REGION Network 1: Block description — Sections 1 to 2
   // ▄▄▄▄▄▄▄▄▄▄▄▄▄▄▄▄▄▄▄▄▄▄▄▄▄▄▄▄▄▄▄▄▄  ＳＴＡＮＤＡＲＤ  ▄▄ 
   // 
   // 
   // TITLE:    SUBROUTINE — ANALOG OUTPUT SCALE
   // 
   // 
   // ▀▀▀▀▀▀▀▀▀▀▀▀▀▀▀▀▀▀▀▀▀▀▀▀▀▀▀▀▀▀▀▀▀▀▀▀▀▀▀▀▀▀▀▀ 
   // 
   // ┌──────────────────────────────────────────┐
   // │                                          │
   // │          FC18002 — SOFTWARE MODULE DESIGN SPECIFICATION (SMDS)            │
   // │                                          │
   // │      The PDF version of the SMDS for this module is available online here:        │
   // │              https://psop.uk/pal-smds-fc18002-p               │
   // │                                          │
   // │      It is also available as part of the Project User Defined Documentation,      │
   // │      it can be accessed by selecting this module in the Project Tree          │
   // │      (on the left) and pressing SHIFT+F1                        │
   // │                                          │
   // └─────────────────────────────────────── ʷᴵᴰ⁻ᵈᶤᵇ  ┘
   // 
   // FC18001_StdSubScaleAI is a subroutine block that is used to convert a scaled device signal to 
   // an integer signal being passed to an analog output in the form of an output word (QW).
   // 
   // The initial scaled value is a real (floating point) number that matches the calibrated range of 
   // the device in engineering units.
   // 
   // The block monitors the scaled signal to see if the scaled value is out-of-range, the following three 
   // fault signals are generated:
   // 
   // 
   //    •   Over-range (signal is more than a specified percentage above the calibrated 
   //      range of the instrument
   // 
   //    •   Under-range (signal is more than a specified percentage below the calibrated 
   //      range of the instrument
   // 
   //    •   Common out-of-range, either the over-range or under-range fault is active
   // 
   // This is a subroutine block.
   // 
   // 
   // 
   // ▄▄▄▄▄▄▄▄▄▄▄▄▄▄▄▄▄▄▄▄▄▄▄▄▄▄▄▄▄▄▄▄▄▄▄▄▄▄▄▄▄▄▄▄
   // 1.     BLOCK TECHNICAL SUMMARY
   // 
   // 
   //  ――――――――――――――――――――――――――――――――――――――――――
   //  NOMENCLATURE & ADDRESSING
   //  ――――――――――――――――――――――――――――――――――――――――――
   //  BLOCK TITLE         Analog Output Scale
   //  BLOCK FUNCTION GROUP    Subroutine
   //  BLOCK ADDRESS       FC18002
   //  BLOCK SYMBOL        FC18002_StdSubScaleAQ
   //  BLOCK USER ID         StdSubScaleAQ
   // 
   //  ――――――――――――――――――――――――――――――――――――――――――
   //  BLOCK TYPE & USAGE
   //  ――――――――――――――――――――――――――――――――――――――――――
   //  BLOCK TYPE         Function (FC)
   //  BLOCK NUMBER        18002
   //  LANGUAGE           LAD
   //  OPTIMISED ACCESS     Yes
   //  PAL USAGE TYPE       Standard block
   // 
   //  ――――――――――――――――――――――――――――――――――――――――――
   //  METRICS
   //  ――――――――――――――――――――――――――――――――――――――――――
   //  EXECUTION TIME       23.6 μs¹
   //  LOAD MEMORY       30.5 kB
   //  WORK MEMORY           0.5 kB  
   //  ――――――――――――――――――――――――――――――――――――――――――
   //                ¹ Measured on: CPU-1515-2PN (order no. 6ES7512-2AM02-0AB0) 
   //                             https://psop.uk/pal-ds-cpu1515
   // 
   // 
   // 
   // ▂▂▂▂▂▂▂▂▂▂▂▂▂▂▂▂▂▂▂▂▂▂▂▂▂▂▂▂▂▂▂▂▂▂▂▂▂▂▂▂▂▂▂▂
   // Additional document references
   // 
   // 
   // In addition to the documents referenced in OB1 (section DOCUMENT REFERENCES), the 
   // following documents are associated with this module:
   // 
   // 
   //  ――――――――――――――――――――――――――――――――――――――――――
   //  REF.     DOCUMENT NO.       TITLE
   //  ――――――――――――――――――――――――――――――――――――――――――
   //  101  PS2001-5-2312-db00801   DB00802 (analog output raw data) SMDS
   //  102  PS2001-5-2312-db00851   DB00852 (analog output scale data) SMDS
   //  ――――――――――――――――――――――――――――――――――――――――――
   // 
   //                ━━━   ⬙⬙⬙⬙⬙⬙   ━━━
   // 
   // 
   // 
   // ▄▄▄▄▄▄▄▄▄▄▄▄▄▄▄▄▄▄▄▄▄▄▄▄▄▄▄▄▄▄▄▄▄▄▄▄▄▄▄▄▄▄▄▄
   // 1.     FUNCTIONAL DESCRIPTION
   // 
   // 
   // FC18002 is the Analog Output Scale block, it is a subroutine block designed to convert a scaled 
   // signal into a form suitable for an analog output it provides the following broad functions:
   // 
   //    •   Converts a scaled, floating point (real) number that reflects the output range of a 
   //      device, into a raw integer signal for an analog output 
   // 
   //    •   Generate fault signals if the instrument is out of range
   // 
   // 
   // 
   // ▂▂▂▂▂▂▂▂▂▂▂▂▂▂▂▂▂▂▂▂▂▂▂▂▂▂▂▂▂▂▂▂▂▂▂▂▂▂▂▂▂▂▂▂
   // 1.1     Convert a scaled value into an analog output
   // 
   // 
   // The principal function of the block is to convert a scaled, floating point (real) number that reflects 
   // the output range of a device, into a raw integer signal for an analog output (in the form of an 
   // output word, QW).
   // 
   // For example, if a variable speed drive had a scaled operating range of 150 rpm to 1500 rpm and 
   // was driven via a 4-20 mA analog output signal from the PLC, then 4 mA would represent 150 rpm 
   // and 20 mA would represent 1500 rpm.
   // 
   // A typical 4-20 mA analog output signal has a raw value of 0 at 4 mA and 27648 at 20 mA.
   //  
   // The block would generate output values as follows (it would also return every value in between; 
   // five typical values have been shown):
   // 
   // 
   //  ――――――――――――――――――――――――――――――――――――――――――
   //  SCALED OUTPUT SIGNAL   RAW INTEGER VALUE FOR OUTPUT   ACTUAL OUTPUT SIGNAL
   //  ――――――――――――――――――――――――――――――――――――――――――
   //     150.0 rpm                     0              4 MA
   //     487.5 rpm             6,912              8 MA
   //     825.0 rpm           13,824            12 MA
   //      1162.5 rpm           20,736            16 MA
   //      1500.0 rpm           27,648            20 MA
   //  ――――――――――――――――――――――――――――――――――――――――――
   // 
   // 
   // 
   // ▂▂▂▂▂▂▂▂▂▂▂▂▂▂▂▂▂▂▂▂▂▂▂▂▂▂▂▂▂▂▂▂▂▂▂▂▂▂▂▂▂▂▂▂
   // 1.2     Fault signals
   // 
   // 
   // The block is able to generate three fault signals:
   // 
   //    •   Device is over-range
   // 
   //    •   Device is under-range
   // 
   //    •   Device is out-of-range (common signal)
   // 
   // Over-range and under-range faults are generated if the device is reading outside its normal 
   // calibrated range. Over-range if the device is reading higher than its maximum configured value 
   // and under-range if lower than its minimum configured value.
   // 
   // The levels at which the device is considered to be either over-range or under-range (out-of-range), 
   // are set as configurable values passed to the module.
   // 
   // The out-of-range fault signal is a common signal that activates if either the over-range or 
   // under-range signal is 
   // 
   // All three signal activate if there is a configuration error with the data provided to the 
   // module (see § 2.1.2).
   // 
   // 
   // 
   // ▄▄▄▄▄▄▄▄▄▄▄▄▄▄▄▄▄▄▄▄▄▄▄▄▄▄▄▄▄▄▄▄▄▄▄▄▄▄▄▄▄▄▄▄
   // 2.     DETAILED BLOCK DESCRIPTION
   // 
   // 
   // This module, FC18001_StdSubScaleAI is a subroutine block that can be called from other blocks 
   // within the PAL. It is designed to provide a linear conversion of a scaled device output signal in 
   // engineering units (in real format) to an integer value that repre-sents the analog output value 
   // passed to an analog output card (as an integer).
   // 
   // These are the formal module parameters: 
   // 
   // 
   // 
   //  ――――――――――――――――――――――――――――――――――――――――――
   //  PARAM          FUNCTION                      TYPE      IN-OUT 
   //  ――――――――――――――――――――――――――――――――――――――――――
   //  AQ_SCALE_SIGNAL   The scaled value of the device output in       Real      In
   //            engineering units
   // 
   //  AQ_RAW_DATA     Analog output signal configuration data (type,     UT00802    In
   //            range, descriptions card parameters and 
   //            coefficients)
   // 
   //  AQ_SCALE_DATA    Analog output signal scaled value data        UT00852   In
   //            (instrument tag, range, descriptions and 
   //            engineering units)
   // 
   //  AQ_RAW_SIGNAL       The actual analog output             Word     Out
   //            engineering units
   // 
   //  OVER_RANGE       Indicates the scaled signal is above its         Bool      Out
   //            calibrated range by more than the tolerance
   //            value
   // 
   //  UNDER_RANGE     Indicates the scaled signal is below its         Bool      Out
   //            calibrated range by more than the tolerance 
   //            value
   // 
   //  OUT_OF_RANGE      Indicates the scaled signal is outside of its     Bool      Out
   //            calibrated range either over or under range
   //  ――――――――――――――――――――――――――――――――――――――――――
   //  Note:   If a configuration error is present (see § 2.1.2) the three out of range parameters 
   //      will be activated (set true) and the AI_SCALE_SIGNAL signal will be set to zero 
   //      irrespective of the AI_RAW_SIGNAL value.
   // 
   // 
   // The AQ_SCALE_SIGNAL signal is provided directly from the module controlling the device and is 
   // a real number in engineering units (e.g. 1220.4 rpm).
   // 
   // The AQ_RAW_SIGNAL signal is the integer value passed directly to the specific output channel 
   // of the analog output card.
   // 
   // The AQ_RAW_DATA and AQ_SCALE_DATA parameters are UDTs that hold information about the 
   // nature of the AQ_RAW_SIGNAL. In the case of AQ_RAW_DATA it specifies the output type: 
   // voltage, current &c., its range in integer values, various par-ametric information and a textual 
   // description of the signal. In the case of AQ_SCALE_DATA it specifies the scaled range of the 
   // signal, its engineering units, out-of-range values, a textual description of the device and the 
   // device tag itself.
   // 
   // 
   //  ――――――――――――――――――――――――――――――――――――――――――
   //  PARAM         ASSOCIATED UDT            ASSOCIATED DATA BLOCK
   //  ――――――――――――――――――――――――――――――――――――――――――
   //  AQ_RAW_DATA    UT00802_St_ConstAqRawData     DB00802_St_ConstAqRawData
   //  AQ_SCALE_DATA   UT00852_St_ConstAqScaleData      DB00852_St_ConstAqScaleData
   //  ――――――――――――――――――――――――――――――――――――――――――
   // 
   // Section 2.1.1 contains a full description of the AQ_RAW_DATA and AQ_SCALE_DATA parameters.
   // 
   // AQ_SCALE_SIGNAL is the true scaled value of the signal being passed to the analog output 
   // (AQ_RAW_SIGNAL) in engineering units.
   // 
   // OVER_RANGE and UNDER_RANGE indicate if the scaled signal is outside its permitted range. 
   // The limits at which under-range and over-range faults activate are provided as part of the 
   // information supplied via the AQ_SCALE_DATA parameter.
   // 
   // OVER_RANGE indicates the output is higher than the permitted tolerance and UNDER_RANGE 
   // indicates the output is lower than the permitted tolerance.
   // 
   // OUT_OF_RANGE is simply a common signal indicating the either OVER_RANGE or UNDER_RANGE 
   // is active.
   // 
   // This arrangement conforms with the PAL philosophy where IO card connections, safety signals 
   // and interlocks have unique formal parameters; all remaining signals are passed as variables 
   // within UDTs, see the Software Design Specification [Ref 008].
   // 
   // 
   // 
   // ▂▂▂▂▂▂▂▂▂▂▂▂▂▂▂▂▂▂▂▂▂▂▂▂▂▂▂▂▂▂▂▂▂▂▂▂▂▂▂▂▂▂▂▂
   // 2.1     Converting the scaled device signal to an analog output value
   // 
   // 
   // The AQ_RAW_SIGNAL is the raw device signal passed to the analog output card; this has specific 
   // ranges depending on the type of IO card and the type of signal in use. 
   //  
   // The following table shows example ranges for the AI_RAW_SIGNAL signal:
   // 
   //  ―――――――――――――――――――――――――――――――――――――――――― 
   //             LOWER LIMIT    EQUIVALENT UPPER LIMIT   EQUIVALENT
   //  SIGNAL TYPE      (RAW_MIN)         TO    (RAW_MAX)       TO      
   //  ―――――――――――――――――――――――――――――――――――――――――― 
   //  -10 V to 10 V         -27648     -10 V        27648      +10 V      
   //  0 V to 10 V          0       +10 V     27648      +10 V      
   //  1 V to 5 V          0      +1 V        27648     +5 V      
   //  -20 mA to 20 mA       -27648     -20 mA    27648      +20 mA      
   //  0 mA to 20 mA         0        0 mA    27648      +20 mA      
   //  4 mA to 20 mA (2/4w)      0        4 mA    27648      +20 mA      
   //  ――――――――――――――――――――――――――――――――――――――――――
   //  Example ranges for an analog output signal
   // 
   // 
   // The RAW_MIN and the RAW_MAX values in the above tables are the numerical values for the 
   // analog output range; the appropriate values are supplied as the RAW_MIN and RAW_MAX 
   // variables provided in the UDT of parameter AQ_RAW_DATA. (see § 2.1.1 for a full description).
   // 	
   // 
   // The corresponding values for the originating scaled device signal are similarly provided by the 
   // SCALE_MIN and SCALE_MAX values provided in the UDT of parameter AQ_SCALE_DATA 
   // (see § 2.1.1 for a full description).
   // 
   // Thus, if a variable speed drive had a scaled operating range of 150 rpm to 1500 rpm that was 
   // passed from the PLC as a 4 20 mA signal, 
   // 
   // 
   //  ――――――――――――――――――――――――――――――――――――――――――
   //  SIGNAL NAME            FUNCTION                   VALUE
   //  ――――――――――――――――――――――――――――――――――――――――――
   //  AQ_RAW_DATA.RAW_MIN     RANGE — Minimum value of the raw analog      0
   //                       signal (at the card)
   //  AQ_RAW_DATA.RAW_MAX    RANGE — Maximum value of the raw analog        27648
   //                       signal (at the card)
   //  AQ_SCALE_DATA.SCALE_MIN   RANGE — Minimum value of the scaled analog       150 rpm
   //                       signal [engineering units]
   //  AQ_SCALE_DATA.SCALE_MAX  RANGE — Maximum value of the scaled analog      1500 rpm
   //                       signal [engineering units]
   //  ――――――――――――――――――――――――――――――――――――――――――
   // 
   // The scaled value from the originating device is passed to the module as a real number in the 
   // parameter: AQ_SCALE_SIGNAL
   // 
   // The analog output signal (AQ_RAW_SIGNAL) is calculated as follows:
   // 
   // 
   // ┌────────────────────────────────────────────┐
   // │                                 (AQ_SCALE_SIGNAL ─ SCALE_MIN) ╳ (RAW_MAX ─ RAW_MIN)         │
   // │AQ_RAW_SIGNAL =  ――――――――――――――――――――――――――――  ┼ RAW_MIN      │
   // │                                    (SCALE_MAX ─ SCALE_MIN)                  │
   // └──────────────────────────────────────  (2.1)  ───┘
   // 
   // In the above calculation, RAW_MIN and RAW_MAX are preceded by AQ_RAW_DATA. and SCALE_MIN and 
   // SCALE_MAX are preceded by AQ_SCALE_DATA.
   // 
   // The three signals: AQ_SCALE_SIGNAL, SCALE_MIN and SCALE_MAX are all floating-point numbers 
   // (real data type), the signals AQ_RAW_SIGNAL, RAW_MIN and RAW_MAX are all integers (int data type).
   // 
   // Note:    It is assumed that the instrument has a linear response.
   // 
   // 
   //           AQ_ SCALE_VALUE
   //             ↑                    ⋰
   //            SCALE_MAX__│______________________________________⋰
   //             │                  ╱|
   //             │                 ╱ |     
   //             │                ╱  |
   //             │               ╱   |
   //             │              ╱    |
   //             │             ╱     |
   //             │            ╱      |
   //     AQ_SCALE_SIGNAL │- - - - - - - - - - - - - - - - - - - - -> ╱       |
   //             │          ╱╎          |
   //             │         ╱ ╎       |
   //             │        ╱  ╎       |
   //             │       ╱   ╎       |   
   //             │      ╱    ╎       |
   //             │     ╱     ╎       |
   //             │    ╱         ╎          |
   //             SCALE_MIN__│______╱          ╎          |
   //             │  ⋰|           ╎          |
   //             │ ⋰ |           ↓          |
   //             ┼─────────────────────────→ AQ_RAW_SIGNAL
   //                   |           ╎           |
   //                RAW_MIN        ╎        RAW_MAX
   //                       AQ_RAW_SIGNAL
   // 
   //    Figure 2.1    Linear relationship between AQ_SCALE_SIGNAL and AQ_RAW_SIGNAL
   // 
   // 
   // 
   // ▁▁▁▁▁▁▁▁▁▁▁▁▁▁▁▁▁▁▁▁▁▁▁▁▁▁▁▁▁▁▁▁▁▁▁▁▁▁▁▁▁▁▁▁
   // 2.1.1     Using AQ_RAW_DATA and AQ_SCALE_DATA
   // 
   // 
   // 
   // ▁▁▁▁▁▁▁▁▁▁▁▁▁▁▁▁▁▁▁▁▁▁▁▁▁▁▁▁▁▁▁▁▁▁▁▁▁▁▁▁▁▁▁▁
   // The AQ_RAW_DATA parameter
   // 
   // The parameter AQ_RAW_DATA is used to pass the analog output card type, range, and description 
   // data used by all analog output card channels. Data is supplied to this parameter using
   // DB00802_St_ConstAqRawData, this contains a formal set of data for every type of Siemens 
   // analog output (datasets), E.g.: for a 4-wire 4-20 mA signal it is:
   // 
   //  AQ_RAW_2002      "UT00802_St_ConstAqRawData" AQ Current (4 mA to 20 mA)
   //   revInfo          "UT01000_St_SysRevision"
   //   ___________0010_0  Bool     false	 
   //   ___________0010_1  Bool     false
   //   AQ_CODE        UInt      16#2002
   //   ___________0020_0  Bool     false
   //   ___________0020_1  Bool     false
   //   RAW_MIN          Int        0
   //   RAW_MAX         Int        27648
   //   RAW_DESC       String[60]    'Current (4 mA to 20 mA)'
   //   ___________0030_1  Bool     false
   //   ___________0030_2  Bool     false
   //   PARAM_TYPE       Byte        16#02
   //   PARAM_RANGE      Byte        16#02
   // 
   // A full description of DB00801_St_ConstAiRawData and its associated datasets is given in 
   // [Ref. 101].
   // 
   // The primary in formation needed by the module are maximum and minimum ranges for the 
   // input signal, this information is given in in the variables:
   // 
   // 
   //  AQ_RAW_DATA
   //  ――――――――――――――――――――――――――――――――――――――――――
   //  SIGNAL NAME           FUNCTION                    TYPE
   //  ――――――――――――――――――――――――――――――――――――――――――
   //  AQ_RAW_DATA.RAW_MIN       Minimum value of the analog input           Int
   //                range being used by the module
   // 
   //  AQ_RAW_DATA.RAW_MAX      Maximum value of the analog input           Int
   //                range being used by the module
   //  ――――――――――――――――――――――――――――――――――――――――――
   // 
   // These are the RAW_MIN and RAW_MAX values used in equation (2.1).
   // 
   // 
   // 
   // ▁▁▁▁▁▁▁▁▁▁▁▁▁▁▁▁▁▁▁▁▁▁▁▁▁▁▁▁▁▁▁▁▁▁▁▁▁▁▁▁▁▁▁▁
   // The AQ_SCALE_DATA parameter
   // 
   // 
   // The AQ_SCALE_DATA parameter is similar to the AI_RAW_DATA parameter except that in this 
   // case it holds the scaled range, instrument tag, signal description and as-sociated engineering 
   // unit information. Data is supplied to this parameter using DB00852_St_ConstAqScaleData, this 
   // contains a set of data each device configured for the project, each device being a 
   // dataset. E.g.
   // 
   //  AQ_SCALE_FC001    "UT00852_Sy_ConstAqScaleData"	
   //   revInfo        "UT01000_St_SysRevision"	
   //   ___________0010_0  Bool     false
   //   ___________0010_1  Bool     false
   //   AQ_TAG         String[20]    'FC001'
   //   ___________0020_0  Bool     false
   //   ___________0020_1  Bool     false
   //   SCALE_MIN         Real        0.0
   //   SCALE_MAX        Real        100.0
   //   SCALE_UNITS     String[20]    '%'
   //   SCALE_DESC      String[60]    'Inlet flow control valve (0 to 100%)'
   //   ___________0030_0  Bool     false
   //   ___________0030_1  Bool     false
   //   LIMIT_UNDER      Real        -2.2     
   //   LIMIT_OVER        Real        102.5     
   //   ___________0040_0  Bool     false
   //   ___________0040_1  Bool     false
   //   USER_INFO_1       String[60]    'Instrument Manufacturer: Siemens'
   //   USER_INFO_2       String[60]    'Instrument type: 2-port magnetic'
   //   USER_INFO_3       String[60]    'Instrument part no.: MXG461.15-0.6'
   //   USER_INFO_4       String[60]    'Instrument serial no.:2075181118'
   //   USER_INFO_5       String[60]    ''
   // 
   // 
   // A full description of DB00852_St_ConstAqScaleData and its application is given in [Ref. 102].
   // 
   // The primary in formation needed by the module are maximum and minimum ranges for the 
   // scaled signal, this information is given in in the AI_SCALE_DATA parameter:
   // 
   // 
   //  ――――――――――――――――――――――――――――――――――――――――――
   //  SIGNAL NAME            FUNCTION                    TYPE
   //  ――――――――――――――――――――――――――――――――――――――――――
   //  AQ_SCALE_DATA.SCALE_MIN      Minimum value of the analog input           Real
   //                 range being used by the module
   // 
   //  AQ_SCALE_DATA.SCALE_MAX     Maximum value of the analog input           Real
   //                 range being used by the module
   //  ――――――――――――――――――――――――――――――――――――――――――
   // 
   // These are the SCALE_MIN and SCALE_MAX values used in (2.1).
   // 
   // Additionally, the instrument tag is contained in the variable 
   // 
   //  ――――――――――――――――――――――――――――――――――――――――――
   //  SIGNAL NAME            FUNCTION                   TYPE
   //  ――――――――――――――――――――――――――――――――――――――――――
   //  AQ_SCALE_DATA.AQ_TAG      Tag name of the device             String[20]
   //  ――――――――――――――――――――――――――――――――――――――――――
   // 
   // 
   // 
   // ▁▁▁▁▁▁▁▁▁▁▁▁▁▁▁▁▁▁▁▁▁▁▁▁▁▁▁▁▁▁▁▁▁▁▁▁▁▁▁▁▁▁▁▁
   // 2.1.2     Configuration errors
   // 
   // 
   // The block requires that both the RAW_MAX/MIN and SCALE_MAX/MIN signals conform to certain 
   // rules:
   // 
   //    1.  RAW_MIN must be less than, and not equal to RAW_MAX
   //    2.  SCALE_MIN must be less than, and not equal to SCALE_MAX
   // 
   // Should either of these conditions not be met, the three out of range parameters will all 
   // be activated (set true) 
   // 
   //      OVER_RANGE
   //      UNDER_RANGE
   //      OUT_OF_RANGE
   // 
   // In addition, the AQ_RAW_SIGNAL signal will be set to zero irrespective of the AQ_SCALE_SIGNAL 
   // value.
   // 
   // 
   // 
   // ▂▂▂▂▂▂▂▂▂▂▂▂▂▂▂▂▂▂▂▂▂▂▂▂▂▂▂▂▂▂▂▂▂▂▂▂▂▂▂▂▂▂▂▂
   // 2.2     Out of range signals
   // 
   // 
   // If the AQ_SCALE_SIGNAL signal is outside the SCALE_MIN to SCALE_MAX range (red dotted area 
   // of the graph, Figure 2.1), the AQ_RAW_VALUE will still be calculated correctly; however, an 
   // appropriate, OVER_RANGE or UNDER_RANGE signal will be generated to indicate that the 
   // AQ_SCALE_SIGNAL signal is outside the calibrated range of the instrument and is potentially no 
   // longer accurate.
   // 
   // Some tolerance is permitted before the OVER_RANGE and UNDER_RANGE signals are activated 
   // (most devices are tolerant of slight over and under shoot readings).
   // 
   // The limits at which an over-range or under-range signal is generated is specified in the dataset 
   // passed to the module in the AQ_SCALE_DATA parameter. Each such dataset is stored in 
   // DB00852_St_ConstAqScaleData (see § 2.1.1) in the variables LIMIT_OVER and LIMIT_UNDER 
   // respectively. These represent the highest and lowest values that the scaled instrument value 
   // can read without being either over-range or under-range:
   // 
   //  AQ_SCALE_DATA
   //  ―――――――――――――――――――――――――――――――――――――――――― 
   //  SIGNAL NAME          FUNCTION                     TYPE
   //  ――――――――――――――――――――――――――――――――――――――――――
   //  LIMIT_UNDER        Lower limit of the scaled instrument value in      Real
   //               engineering units before instrument is 
   //               under-range
   // 
   //  LIMIT_OVER           Upper limit of the scaled instrument value in      Real
   //               engineering units before instrument is 
   //               over-range
   //  ――――――――――――――――――――――――――――――――――――――――――
   // 
   // 
   // 
   // ▁▁▁▁▁▁▁▁▁▁▁▁▁▁▁▁▁▁▁▁▁▁▁▁▁▁▁▁▁▁▁▁▁▁▁▁▁▁▁▁▁▁▁▁
   // 2.2.1     Common out of range signal
   // 
   // 
   // There is a third out of range signal: OUT_OF_RANGE, this signal is a common signal that just 
   // indicates the device is out of its calibrated range (it does not specify whether it is over or 
   // under range). 
   // 
   // It is activated if either the OVER_RANGE or UNDER_RANGE signal is active.
   // 
   // Note:    If a configuration error exists, see § 2.1.2, all three out of range signals (OVER_RANGE, 
   //      UNDER_RANGE and OUT_OF_RANGE) will be activated irrespective of the 
   //      RAW_ANALOG value
   // 
   // 
   // 
   // ▁▁▁▁▁▁▁▁▁▁▁▁▁▁▁▁▁▁▁▁▁▁▁▁▁▁▁▁▁▁▁▁▁▁▁▁▁▁▁▁▁▁▁▁
   // 2.2.2    Over and under range restrictions
   // 
   // 
   // The out-of-range limits passed to the module (AQ_SCALE_DATA) must meet the following 
   // conditions:
   // 
   //    •   LIMIT_UNDER ≤ SCALE_MIN
   //    •   LIMIT_OVER ≥ SCALE_MAX
   // 
   // I.e. the device cannot be considered either under range or over range if it is within the 
   // normal range of the device.
   // 
   // If the over-range limit (LIMIT_OVER) is less than SCALE_MAX, then it’s value will be replaced by 
   // SCALE_MAX in all calculations. Similarly, if the under-range limit (LIMIT_UNDER) is greater than 
   // SCALE_MIN, then it’s value will be replaced by SCALE_MIN in all calculations.
   // 
   // 
   // 
   //                ━━━   ⬙⬙⬙⬙⬙⬙   ━━━
END_REGION

REGION Network 2: Block description — Sections 3 to 9
   // ▄▄▄▄▄▄▄▄▄▄▄▄▄▄▄▄▄▄▄▄▄▄▄▄▄▄▄▄▄▄▄▄▄▄▄▄▄▄▄▄▄▄▄▄
   // 3.     Supervisory system interface
   // 
   // 
   // FC18002 is a Subroutine block used to scale an analog input. 
   // 
   // It does not have a supervisory system interface.
   // 
   // 
   //                ━━━   ⬙⬙⬙⬙⬙⬙   ━━━
   // 
   // 
   // 
   // ▄▄▄▄▄▄▄▄▄▄▄▄▄▄▄▄▄▄▄▄▄▄▄▄▄▄▄▄▄▄▄▄▄▄▄▄▄▄▄▄▄▄▄▄
   // 4.     PARAMETERS
   // 
   // The following parameters are associated with this module:
   // 
   // 
   //  ――――――――――――――――――――――――――――――――――――――――――
   //  PARAM          FUNCTION                      TYPE      IN-OUT 
   //  ――――――――――――――――――――――――――――――――――――――――――
   //  AQ_SCALE_SIGNAL   The scaled value of the device output in       Real      In
   //            engineering units
   // 
   //  AQ_RAW_DATA     Analog output signal configuration data (type,     UT00802    In
   //            range, descriptions card parameters and 
   //            coefficients)
   // 
   //  AQ_SCALE_DATA    Analog output signal scaled value data        UT00852   In
   //            (instrument tag, range, descriptions and 
   //            engineering units)
   // 
   //  AQ_RAW_SIGNAL       The actual analog output             Word     Out
   //            engineering units
   // 
   //  OVER_RANGE       Indicates the scaled signal is above its         Bool      Out
   //            calibrated range by more than the tolerance
   //            value
   // 
   //  UNDER_RANGE     Indicates the scaled signal is below its         Bool      Out
   //            calibrated range by more than the tolerance 
   //            value
   // 
   //  OUT_OF_RANGE      Indicates the scaled signal is outside of its     Bool      Out
   //            calibrated range either over or under range
   //  ――――――――――――――――――――――――――――――――――――――――――
   //  Note:   If a configuration error is present (see § 2.1.2) the three out of range parameters 
   //      will be activated (set true) and the AI_SCALE_SIGNAL signal will be set to zero 
   //      irrespective of the AI_RAW_SIGNAL value.
   // 
   //                ━━━   ⬙⬙⬙⬙⬙⬙   ━━━
   // 
   // 
   // 
   // ▄▄▄▄▄▄▄▄▄▄▄▄▄▄▄▄▄▄▄▄▄▄▄▄▄▄▄▄▄▄▄▄▄▄▄▄▄▄▄▄▄▄▄▄
   // 5.     DATA STRUCTURES AND USAGE
   // 
   // 
   // The block has the following associated data structure:
   // 
   // 
   //  ――――――――――――――――――――――――――――――――――――――――――
   //  DATA STRUCTURE             DESCRIPTION
   //  ――――――――――――――――――――――――――――――――――――――――――
   //  UT01000_St_SysRevision          Revision information for this block    See FC01001
   //  UT01001_St_SysLicence           Licence information for this block  See FC01001
   // 
   //  UT00802_St_ConstAqRawData      Analog output signal configuration data 
   //                     (type, range, descriptions card parameters &c.)
   // 
   //  UT00852_St_ConstAqScaleData       Analog output signal scaled value data 
   //                     (instrument tag, range, descriptions and 
   //                     engineering units)
   //  ――――――――――――――――――――――――――――――――――――――――――
   //  Note:   This subroutine does not require the system signals data interface 
   //         (DB21001_Dy_SysSignals). The module is entirely autonomous.
   // 
   // 
   // 
   // ▂▂▂▂▂▂▂▂▂▂▂▂▂▂▂▂▂▂▂▂▂▂▂▂▂▂▂▂▂▂▂▂▂▂▂▂▂▂▂▂▂▂▂▂
   // 5.1     UT00802_St_ConstAqRawData
   // 
   // 
   // The static data structure for an analog instrument.
   // 
   // 
   //  UT00802_St_ConstAqRawData (full contents)
   //  ―――――――――――――――――――――――――――――――――――――――――― 
   //  SIGNAL NAME          FUNCTION                     TYPE
   //  ――――――――――――――――――――――――――――――――――――――――――
   //  AQ_CODE             A 16-bit hex value that uniquely identifies dataset   UInt
   //               (it is the variable name of the dataset in DB00802)
   //  RAW_MIN         Minimum value of the raw analog signal        Int
   //               (at the card)
   // 
   //  RAW_MAX           Maximum value of the raw analog signal        Int
   //  RAW_DESC         Textual plain English description of the channel     String[60]
   //               type and range
   //  PARAM_TYPE         An 8-bit hex code that represents the input type    Byte
   //               See [Ref. 101]
   // 
   //  PARAM_RANGE        An 8-bit hex code that represents the input range    Byte
   //               See [Ref. 101]
   // 
   //  ―――――――――――――――――――――――――――――――――――――――――― 
   // 
   // 
   // 
   // ▂▂▂▂▂▂▂▂▂▂▂▂▂▂▂▂▂▂▂▂▂▂▂▂▂▂▂▂▂▂▂▂▂▂▂▂▂▂▂▂▂▂▂▂
   // 5.2     UT00852_St_ConstAqScaleData
   // 
   // 
   // The static data structure for an analog instrument.
   // 
   // 
   //  UT00852_St_ConstAqScaleDataa (full contents)
   //  ―――――――――――――――――――――――――――――――――――――――――― 
   //  SIGNAL NAME          FUNCTION                     TYPE
   //  ――――――――――――――――――――――――――――――――――――――――――
   //  AQ_TAG           Tag name of the instrument             String[20]
   // 
   //  SCALE_MIN        Minimum value of the scaled input signal range    Real
   //               being used by the module
   //  SCALE_MAX          Maximum value of the scaled input signal range      Real
   //               being used by the module
   // 
   //  SCALE_UNITS          Engineering units for the instrument         String[20]
   //  SCALE_DESC           Textual plain English description of the instrument  String[60]
   // 
   //  LIMIT_UNDER        Lower limit of the scaled instrument value in      Real
   //               engineering units before instrument is 
   //               under-range
   //  LIMIT_OVER           Upper limit of the scaled instrument value in      Real
   //               engineering units before instrument is 
   //               over-range
   // 
   //  USER_INFO_1          Optional user information (text) line 1       String[60]
   //  USER_INFO_2          Optional user information (text) line 2       String[60]
   //  USER_INFO_3          Optional user information (text) line 3       String[60]
   //  USER_INFO_4          Optional user information (text) line 4       String[60]
   //  USER_INFO_5          Optional user information (text) line 5       String[60]
   //  ―――――――――――――――――――――――――――――――――――――――――― 
   // 
   //                ━━━   ⬙⬙⬙⬙⬙⬙   ━━━
   // 
   // 
   // 
   // 
   // ▄▄▄▄▄▄▄▄▄▄▄▄▄▄▄▄▄▄▄▄▄▄▄▄▄▄▄▄▄▄▄▄▄▄▄▄▄▄▄▄▄▄▄▄
   // 6.     CONSTANTS AND TEMPORARY (LOCAL) DATA
   // 
   // 
   // 
   // ▂▂▂▂▂▂▂▂▂▂▂▂▂▂▂▂▂▂▂▂▂▂▂▂▂▂▂▂▂▂▂▂▂▂▂▂▂▂▂▂▂▂▂▂
   // 6.1     Constants
   // 
   // 
   // No constants are used in this block.
   // 
   // 
   // 
   // ▂▂▂▂▂▂▂▂▂▂▂▂▂▂▂▂▂▂▂▂▂▂▂▂▂▂▂▂▂▂▂▂▂▂▂▂▂▂▂▂▂▂▂▂
   // 6.2     Temporary (local) data
   // 
   // 
   // The following temporary data is used:
   // 
   //  ――――――――――――――――――――――――――――――――――――――――――
   //  SIGNAL NAME          FUNCTION                    TYPE
   //  ――――――――――――――――――――――――――――――――――――――――――
   //  revInfo             Revision information for the block           UT01000
   //  licInfo           Licensing information for the block        UT01001
   //  calPart1             Raw value part 1 (SCALE_ANALOG − SCALE_MIN)       Real
   //  calPart2             Raw value part 2 (SCALE_MAX − SCALE_MIN)        Real
   //  calPart3             Raw value part 3 (RAW_MAX − RAW_MIN)      Real
   //  wrkLimitUnder        Actual LIMIT_UNDER in use            Real
   //  wrkLimitOver          Actual LIMIT_OVER in use              Real
   //  wrkConfigError        Working configuration error exists           Bool
   //  wrkReal           Working storage (Real)               Real
   //  ―――――――――――――――――――――――――――――――――――――――――
   // 
   //                ━━━   ⬙⬙⬙⬙⬙⬙   ━━━
   // 
   // 
   // 
   // 
   // ▄▄▄▄▄▄▄▄▄▄▄▄▄▄▄▄▄▄▄▄▄▄▄▄▄▄▄▄▄▄▄▄▄▄▄▄▄▄▄▄▄▄▄▄
   // 7.     BLOCK CALLS AND ASSOCIATIONS
   // 
   // 
   // This section details any blocks which may be called from within this software module (subroutine 
   // functions for example), any partner blocks with which it may be associated (for example a 
   // receive module that is partner with a transmit module &c.). It lists any system functions which 
   // may be called (e.g. reading the real time clock) and any system data types that may be used.
   // 
   // Finally, it lists any special calling requirements for the block (for example, must be called from 
   // within a cyclic interrupt organisation block) and if the block is using “optimised access” (this is 
   // the default arrangement).
   // 
   // 
   // 
   // ▂▂▂▂▂▂▂▂▂▂▂▂▂▂▂▂▂▂▂▂▂▂▂▂▂▂▂▂▂▂▂▂▂▂▂▂▂▂▂▂▂▂▂▂
   // 7.1     Block calls from within this module
   // 
   // 
   // There are no PAL block calls from within this block.
   // 
   // 
   // 
   // ▂▂▂▂▂▂▂▂▂▂▂▂▂▂▂▂▂▂▂▂▂▂▂▂▂▂▂▂▂▂▂▂▂▂▂▂▂▂▂▂▂▂▂▂
   // 7.2     Blocks associated with this module
   // 
   // 
   // This is a stand-alone block and is not associated with any other blocks.
   // 
   // 
   // 
   // ▂▂▂▂▂▂▂▂▂▂▂▂▂▂▂▂▂▂▂▂▂▂▂▂▂▂▂▂▂▂▂▂▂▂▂▂▂▂▂▂▂▂▂▂
   // 7.3     System block calls and system data types
   // 
   // There are no system block calls
   // 
   // 
   // 
   // ▂▂▂▂▂▂▂▂▂▂▂▂▂▂▂▂▂▂▂▂▂▂▂▂▂▂▂▂▂▂▂▂▂▂▂▂▂▂▂▂▂▂▂▂
   // 7.4     Special properties and requirements
   // 
   // 
   // 
   // ▁▁▁▁▁▁▁▁▁▁▁▁▁▁▁▁▁▁▁▁▁▁▁▁▁▁▁▁▁▁▁▁▁▁▁▁▁▁▁▁▁▁▁▁
   // 7.4.1     Block optimisation, IEC compatibility and library conformance
   // 
   // 
   //    •   Block optimisation is ACTIVE for this block.
   // 
   //    •   The block has been checked for IEC compatibility and is compliant.
   // 
   //    •   The block is compatible with all IEC library-conformance module constraints
   // 
   // 
   // 
   // ▁▁▁▁▁▁▁▁▁▁▁▁▁▁▁▁▁▁▁▁▁▁▁▁▁▁▁▁▁▁▁▁▁▁▁▁▁▁▁▁▁▁▁▁
   // 7.4.2     Calling requirements
   // 
   // 
   // There are no special calling requirements for this block.
   // 
   //                ━━━   ⬙⬙⬙⬙⬙⬙   ━━━
   // 
   // 
   // 
   // ▄▄▄▄▄▄▄▄▄▄▄▄▄▄▄▄▄▄▄▄▄▄▄▄▄▄▄▄▄▄▄▄▄▄▄▄▄▄▄▄▄▄▄▄
   // 8.     EXAMPLE USAGE
   // 
   // 
   // The following shows a typical deployment of FC18002:
   // 
   // 
   //                        ┌─────────────
   //         ───────────────┤ FC18002
   //                        ├───────────
   //                        │              │                       
   //                           "FCV001"   ─┤ AQ_SCALE_SIGNAL      │
   //                        │              │
   //        "DB00802".AQ_RAW_2003    ─┤ AQ_RAW_DATA        │
   //                        │              │
   //        "DB00852".AQ_SCALE_FCV001 ─┤ AQ_SCALE_DATA       │
   //                        │              │
   //                             AQ_SCALE_SIGNAL├─ #FCV001_RAW
   //                                    │
   //                              UNDER_RANGE ├─ #ALM_UNDER
   //                                    │
   //                                 OVER_RANGE├─ #ALM_OVER
   //                                    │
   //                                  OUT_OF_RANGE├─ #ALM_OOR  
   //                                    │
   //                       ─────────────┘
   // 
   // 
   //                ━━━   ⬙⬙⬙⬙⬙⬙   ━━━
   // 
   // 
   // 
   // ▄▄▄▄▄▄▄▄▄▄▄▄▄▄▄▄▄▄▄▄▄▄▄▄▄▄▄▄▄▄▄▄▄▄▄▄▄▄▄▄▄▄▄▄
   // 9.     TEST AND VERIFICATION PATH
   // 
   // 
   // The following diagram shows the full test and verification path for the formal release of each 
   // version of the software module. See the Test Plan [Ref. 003] for full details, available here:
   //         https://psop.uk/pal-tp-p
   // 
   // 
   //         FC18002-T001   
   // 
   //     Test version: 000.801     
   //  Released version: 001.000     
   // Released commit: D0018    
   // 
   //        SCR      SMT  
   // ＿＿＿＿＿＿┌┐＿＿ ▛▜ ＿＿
   //       └┘   ▙▟   
   // Initial test           
   // 
   // Initial test to release the      
   // module following the      
   // development stage.       
   // Full SMT              
   //                             
   // 
   // Where:
   // ――――――――――――――――――――――――――――――――――――――――――――
   //  SCR    Source Code Review      A visual inspection of the software to ensure it has been written  
   // ┌┐             to the correct standards, uses the correct structures within the
   // └┘             software and is generally suitable for deployment.               
   // 
   //  SMT Software Module Test    A full and detailed test of an individual software module in
   //   ▛▜              isolation; such testing requires that all branches of the 
   //   ▙▟              software are tested. 
   // 
   //                It tests all the interfaces to the module, any data recorded or 
   //                stored by the module, all error and exception handling functions 
   //                and tests all timed and interrupt driven operations.
   // 
   //  SMTp SMT partial retest      A partial repeat of some aspect of the full SMT to retest a small
   //   ▛ ┐               change made to some aspect of the software. The change 
   // └ ▟                must be small, specific and localised.
   // 
   //  SCV Software Compatibility     A mechanism for verifying that no executable code software 
   // ╓╖    Verification          changes have been made to a module following changes to
   // ╙╜             comment fields.
   // 
   //                Allows typographical errors &c. to be corrected without forcing 
   //                a full SMT on a module that has not functionally changed.
   // ――――――――――――――――――――――――――――――――――――――――――――
   // 
   // An SCV can only be performed on a module that has at some point previously, successfully 
   // completed both an SCR and SMT. Where an SCV is implemented, it replaces the requirement for 
   // both the SCR and the SMT for the test iteration in question.
   // 
   //                ━━━   ⬙⬙⬙⬙⬙⬙   ━━━
   // 
   // 
   // ██████████████ █ █ █ █  END   █ █ █ █ ██████████████
END_REGION

REGION Network 3: Current revision and modification history
   // ▄▄▄▄▄▄▄▄▄▄▄▄▄▄▄▄▄▄▄▄▄▄▄▄▄▄▄▄▄▄▄▄▄▄▄▄▄▄▄▄▄▄▄▄
   // MODIFICATION HISTORY
   // 
   // 
   // The revision data shown here, in the network comments, contains additional information 
   // reflecting the software development workflow under the version control system (VCS) employed 
   // to track all software changes.
   // 
   // The VCS in use is the Git Source Code Management system in conjunction with the GitHub online 
   // hosting system. The software in its entirety is available in the GitHub remote repository:
   // 
   //      https://github.com/practicalseries/PS2001-pal-software
   // 
   // The repository is public and can be freely copied (forked in GitHub terminology) and used 
   // under the MIT licence. 
   // 
   // The MIT licence is reproduced in full in the last network of this software module.
   // 
   // 
   //  ―――――――――――――――――――――――――――――――――――――――――――
   //  DATE       REVISION             MASTER BRANCH     DEV
   //          (nnn.amm)   COMMIT TAG    (Base ---> Merge)    BRANCH   Author
   //  ———————————————————————————————————————————
   //  2022.09.03    001.000   D0018      D0017 D0018  None    M. Gledhill
   //                        FC18001 — RELEASED FOR USE
   //                          Merge back to master branch
   // 
   //  2024.09.02    000.101   D0017A-000.109   D0017 N/A     D0017A   M. Gledhill
   //                        Block created
   //  ———————————————————————————————————————————
   //   Where: nnn  =  Major revision
   //         a  =  Type (1-7 Development, 8 Proving, 9 Qualification, 0 Release)
   //       mm  =  Minor revision (must be 00 if a = 0)
   //         Block properties version number should be set to nn.a (only one decimal place)
   // 
   // ▄▄▄▄▄▄▄▄▄▄▄▄▄▄▄▄▄▄▄▄▄▄▄▄▄▄▄▄▄▄▄▄▄▄▄▄▄▄▄▄▄▄▄▄
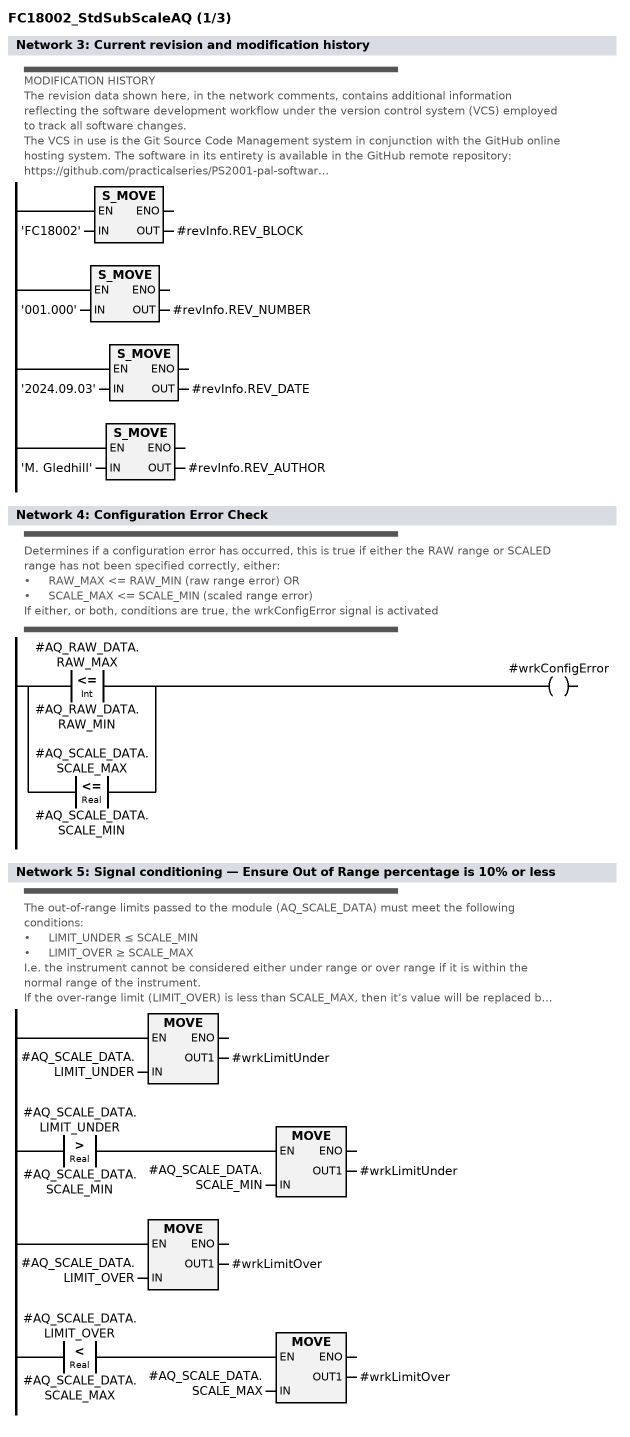
   RUNG wire#powerrail
      S_Move(in := 'FC18002', out => #revInfo.REV_BLOCK)
   END_RUNG
   RUNG wire#powerrail
      S_Move(in := '001.000', out => #revInfo.REV_NUMBER)
   END_RUNG
   RUNG wire#powerrail
      S_Move(in := '2024.09.03', out => #revInfo.REV_DATE)
   END_RUNG
   RUNG wire#powerrail
      S_Move(in := 'M. Gledhill', out => #revInfo.REV_AUTHOR)
   END_RUNG
   // the same network as SCL:
   #revInfo.REV_BLOCK := 'FC18002';
   #revInfo.REV_NUMBER := '001.000';
   #revInfo.REV_DATE := '2024.09.03';
   #revInfo.REV_AUTHOR := 'M. Gledhill';
END_REGION

REGION Network 4: Configuration Error Check
   // ▀▀▀▀▀▀▀▀▀▀▀▀▀▀▀▀▀▀▀▀▀▀▀▀▀▀▀▀▀▀▀▀▀▀▀▀▀▀▀▀▀▀▀▀
   // Determines if a configuration error has occurred, this is true if either the RAW range or SCALED 
   // range has not been specified correctly, either:
   // 
   //    •   RAW_MAX <= RAW_MIN (raw range error) OR
   //    •   SCALE_MAX <= SCALE_MIN (scaled range error)
   // 
   // If either, or both, conditions are true, the wrkConfigError signal is activated
   // ▄▄▄▄▄▄▄▄▄▄▄▄▄▄▄▄▄▄▄▄▄▄▄▄▄▄▄▄▄▄▄▄▄▄▄▄▄▄▄▄▄▄▄▄
   RUNG wire#powerrail
      { S7_Templates := "SrcType := Int" } LE_Contact(in1 := #AQ_RAW_DATA.RAW_MAX, in2 := #AQ_RAW_DATA.RAW_MIN)
      wire#w1
      Coil( #wrkConfigError )
   END_RUNG
   RUNG wire#powerrail
      { S7_Templates := "SrcType := Real" } LE_Contact(in1 := #AQ_SCALE_DATA.SCALE_MAX, in2 := #AQ_SCALE_DATA.SCALE_MIN)
   END_RUNG wire#w1
   // the same network as SCL:
   #wrkConfigError := (#AQ_RAW_DATA.RAW_MAX <= #AQ_RAW_DATA.RAW_MIN) OR (#AQ_SCALE_DATA.SCALE_MAX <= #AQ_SCALE_DATA.SCALE_MIN);
END_REGION

REGION Network 5: Signal conditioning — Ensure Out of Range percentage is 10% or less
   // ▀▀▀▀▀▀▀▀▀▀▀▀▀▀▀▀▀▀▀▀▀▀▀▀▀▀▀▀▀▀▀▀▀▀▀▀▀▀▀▀▀▀▀▀
   // The out-of-range limits passed to the module (AQ_SCALE_DATA) must meet the following 
   // conditions:
   // 
   //    •   LIMIT_UNDER ≤ SCALE_MIN
   //    •   LIMIT_OVER ≥ SCALE_MAX
   // 
   // I.e. the instrument cannot be considered either under range or over range if it is within the 
   // normal range of the instrument.
   // 
   // If the over-range limit (LIMIT_OVER) is less than SCALE_MAX, then it’s value will be replaced by 
   // SCALE_MAX in all calculations. Similarly, if the under-range limit (LIMIT_UNDER) is greater than 
   // SCALE_MIN, then it’s value will be replaced by SCALE_MIN in all calculations.
   // 
   // The limits in use are stored in wrkLimitUnder and wrkLimitOver
   // ▄▄▄▄▄▄▄▄▄▄▄▄▄▄▄▄▄▄▄▄▄▄▄▄▄▄▄▄▄▄▄▄▄▄▄▄▄▄▄▄▄▄▄▄
   RUNG wire#powerrail
      Move(in := #AQ_SCALE_DATA.LIMIT_UNDER, out1 => #wrkLimitUnder)
   END_RUNG
   RUNG wire#powerrail
      { S7_Templates := "SrcType := Real" } GT_Contact(in1 := #AQ_SCALE_DATA.LIMIT_UNDER, in2 := #AQ_SCALE_DATA.SCALE_MIN)
      Move(in := #AQ_SCALE_DATA.SCALE_MIN, out1 => #wrkLimitUnder)
   END_RUNG
   RUNG wire#powerrail
      Move(in := #AQ_SCALE_DATA.LIMIT_OVER, out1 => #wrkLimitOver)
   END_RUNG
   RUNG wire#powerrail
      { S7_Templates := "SrcType := Real" } LT_Contact(in1 := #AQ_SCALE_DATA.LIMIT_OVER, in2 := #AQ_SCALE_DATA.SCALE_MAX)
      Move(in := #AQ_SCALE_DATA.SCALE_MAX, out1 => #wrkLimitOver)
   END_RUNG
   // the same network as SCL:
   #wrkLimitUnder := #AQ_SCALE_DATA.LIMIT_UNDER;
   IF #AQ_SCALE_DATA.LIMIT_UNDER > #AQ_SCALE_DATA.SCALE_MIN THEN
       #wrkLimitUnder := #AQ_SCALE_DATA.SCALE_MIN;
   END_IF;
   #wrkLimitOver := #AQ_SCALE_DATA.LIMIT_OVER;
   IF #AQ_SCALE_DATA.LIMIT_OVER < #AQ_SCALE_DATA.SCALE_MAX THEN
       #wrkLimitOver := #AQ_SCALE_DATA.SCALE_MAX;
   END_IF;
END_REGION

REGION Network 6: IO evaluation — Analog output calculation - Part 1
   // ▀▀▀▀▀▀▀▀▀▀▀▀▀▀▀▀▀▀▀▀▀▀▀▀▀▀▀▀▀▀▀▀▀▀▀▀▀▀▀▀▀▀▀▀
   // The following formula is used to calculate the raw analog output signal (AQ_RAW_SIGNAL):
   // ┌────────────────────────────────────────────┐
   // │                                 (AQ_SCALE_SIGNAL ─ SCALE_MIN) ╳ (RAW_MAX ─ RAW_MIN)         │
   // │AQ_RAW_SIGNAL =  ――――――――――――――――――――――――――――  ┼ RAW_MIN      │
   // │                                    (SCALE_MAX ─ SCALE_MIN)                  │
   // └────────────────────────────────────────────┘
   // 
   // Rawvalue calculation part 1 is (AQ_SCALE_SIGNAL − SCALE_MIN)
   // ▄▄▄▄▄▄▄▄▄▄▄▄▄▄▄▄▄▄▄▄▄▄▄▄▄▄▄▄▄▄▄▄▄▄▄▄▄▄▄▄▄▄▄▄
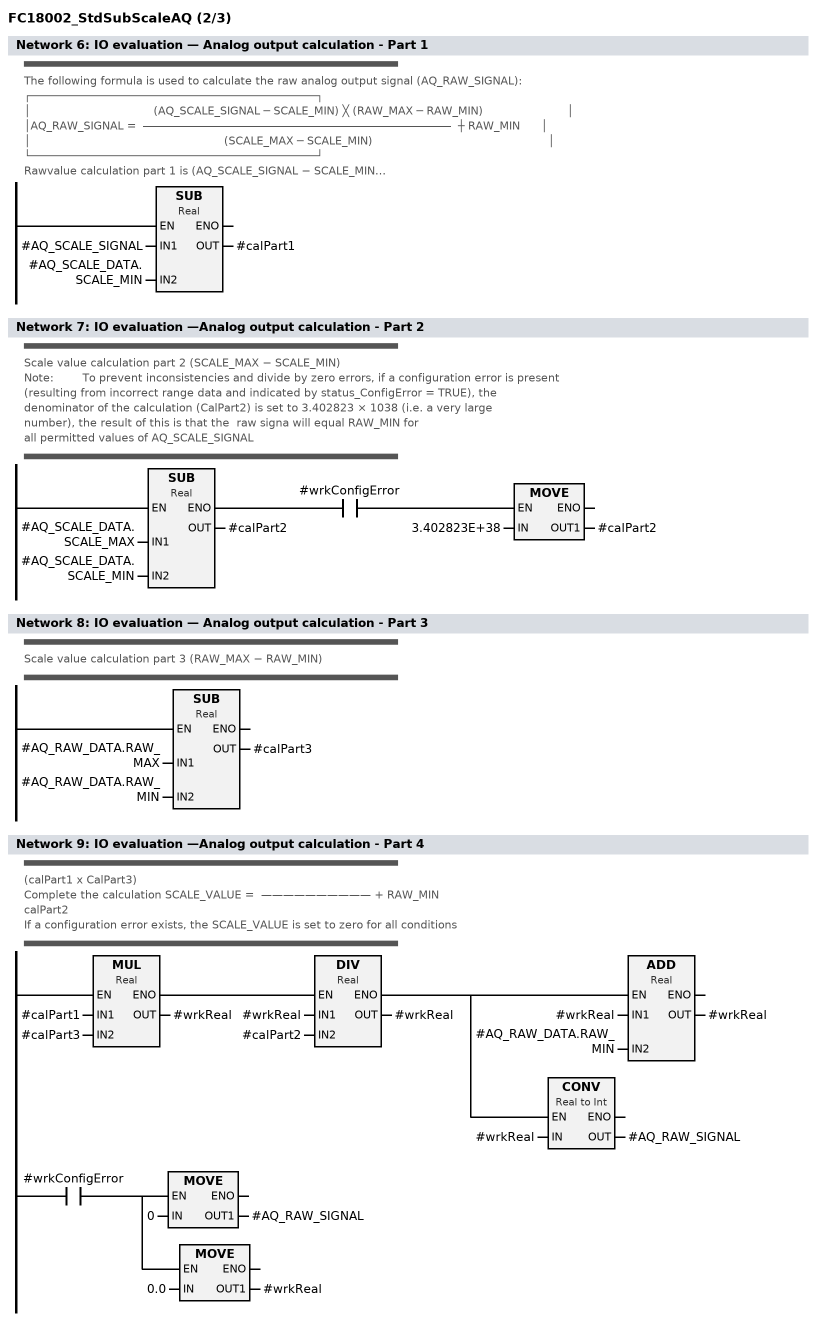
   RUNG wire#powerrail
      { S7_Templates := "SrcType := Real"; S7_GenerateENO := "TRUE" } Sub(in1 := #AQ_SCALE_SIGNAL, in2 := #AQ_SCALE_DATA.SCALE_MIN, out => #calPart1)
   END_RUNG
   // the same network as SCL:
   #calPart1 := #AQ_SCALE_SIGNAL - #AQ_SCALE_DATA.SCALE_MIN;
END_REGION

REGION Network 7: IO evaluation —Analog output calculation - Part 2
   // ▀▀▀▀▀▀▀▀▀▀▀▀▀▀▀▀▀▀▀▀▀▀▀▀▀▀▀▀▀▀▀▀▀▀▀▀▀▀▀▀▀▀▀▀
   // Scale value calculation part 2 (SCALE_MAX − SCALE_MIN)
   // 
   // Note:    To prevent inconsistencies and divide by zero errors, if a configuration error is present
   //      (resulting from incorrect range data and indicated by status_ConfigError = TRUE), the
   //      denominator of the calculation (CalPart2) is set to 3.402823 × 1038 (i.e. a very large 
   //      number), the result of this is that the  raw signa will equal RAW_MIN for 
   //      all permitted values of AQ_SCALE_SIGNAL
   // ▄▄▄▄▄▄▄▄▄▄▄▄▄▄▄▄▄▄▄▄▄▄▄▄▄▄▄▄▄▄▄▄▄▄▄▄▄▄▄▄▄▄▄▄
   RUNG wire#powerrail
      { S7_Templates := "SrcType := Real"; S7_GenerateENO := "TRUE" } Sub(in1 := #AQ_SCALE_DATA.SCALE_MAX, in2 := #AQ_SCALE_DATA.SCALE_MIN, out => #calPart2)
      Contact( #wrkConfigError )
      Move(in := 3.402823E+38, out1 => #calPart2)
   END_RUNG
   // the same network as SCL:
   // ENO of a box is taken as its EN; it also drops when the box reports an error
   #calPart2 := #AQ_SCALE_DATA.SCALE_MAX - #AQ_SCALE_DATA.SCALE_MIN;
   IF #wrkConfigError THEN #calPart2 := 3.402823E+38; END_IF;
END_REGION

REGION Network 8: IO evaluation — Analog output calculation - Part 3
   // ▀▀▀▀▀▀▀▀▀▀▀▀▀▀▀▀▀▀▀▀▀▀▀▀▀▀▀▀▀▀▀▀▀▀▀▀▀▀▀▀▀▀▀▀
   // Scale value calculation part 3 (RAW_MAX − RAW_MIN)
   // ▄▄▄▄▄▄▄▄▄▄▄▄▄▄▄▄▄▄▄▄▄▄▄▄▄▄▄▄▄▄▄▄▄▄▄▄▄▄▄▄▄▄▄▄
   RUNG wire#powerrail
      { S7_Templates := "SrcType := Real"; S7_GenerateENO := "TRUE" } Sub(in1 := #AQ_RAW_DATA.RAW_MAX, in2 := #AQ_RAW_DATA.RAW_MIN, out => #calPart3)
   END_RUNG
   // the same network as SCL:
   #calPart3 := #AQ_RAW_DATA.RAW_MAX - #AQ_RAW_DATA.RAW_MIN;
END_REGION

REGION Network 9: IO evaluation —Analog output calculation - Part 4
   // ▀▀▀▀▀▀▀▀▀▀▀▀▀▀▀▀▀▀▀▀▀▀▀▀▀▀▀▀▀▀▀▀▀▀▀▀▀▀▀▀▀▀▀▀
   //                                                                              (calPart1 x CalPart3)
   // Complete the calculation SCALE_VALUE =  —————————— + RAW_MIN
   //                                                                                         calPart2
   // 
   // If a configuration error exists, the SCALE_VALUE is set to zero for all conditions
   // ▄▄▄▄▄▄▄▄▄▄▄▄▄▄▄▄▄▄▄▄▄▄▄▄▄▄▄▄▄▄▄▄▄▄▄▄▄▄▄▄▄▄▄▄
   RUNG wire#powerrail
      { S7_Templates := "SrcType := Real"; S7_GenerateENO := "TRUE" } Mul(in1 := #calPart1, in2 := #calPart3, out => #wrkReal)
      { S7_Templates := "SrcType := Real"; S7_GenerateENO := "TRUE" } Div(in1 := #wrkReal, in2 := #calPart2, out => #wrkReal)
      wire#w1
      { S7_Templates := "SrcType := Real"; S7_GenerateENO := "TRUE" } Add(in1 := #wrkReal, in2 := #AQ_RAW_DATA.RAW_MIN, out => #wrkReal)
   END_RUNG
   RUNG wire#w1
      { S7_Templates := "[SrcType := Real, DestType := Int]" } Convert(in := #wrkReal, out => #AQ_RAW_SIGNAL)
   END_RUNG
   RUNG wire#powerrail
      Contact( #wrkConfigError )
      wire#w2
      Move(in := 0, out1 => #AQ_RAW_SIGNAL)
   END_RUNG
   RUNG wire#w2
      Move(in := 0.0, out1 => #wrkReal)
   END_RUNG
   // the same network as SCL:
   // ENO of a box is taken as its EN; it also drops when the box reports an error
   #wrkReal := #calPart1 * #calPart3;
   #wrkReal := #wrkReal / #calPart2;
   #wrkReal := #wrkReal + #AQ_RAW_DATA.RAW_MIN;
   #AQ_RAW_SIGNAL := REAL_TO_INT(#wrkReal);
   IF #wrkConfigError THEN
       #AQ_RAW_SIGNAL := 0;
       #wrkReal := 0.0;
   END_IF;
END_REGION

REGION Network 10: IO evaluation — Out of range signals
   // ▀▀▀▀▀▀▀▀▀▀▀▀▀▀▀▀▀▀▀▀▀▀▀▀▀▀▀▀▀▀▀▀▀▀▀▀▀▀▀▀▀▀▀▀
   // The device signal is over range if AQ_SCALED_SIGNAL is greater than wrkLimitOver
   // 
   // The instrument is under range if AQ_SCALED_SIGNAL is less than wrkLimitUnder
   // 
   // If either of these conditions is true, the common out of range signal is activated
   // 
   // Note:    If the range information is incorrect (wrkConfigError = TRUE),
   //      Then all the out of range signals are activated (UNDER_RANGE, 
   //      OVER_RANGE and OUT_OF_RANGE) simultaneously
   // ▄▄▄▄▄▄▄▄▄▄▄▄▄▄▄▄▄▄▄▄▄▄▄▄▄▄▄▄▄▄▄▄▄▄▄▄▄▄▄▄▄▄▄▄
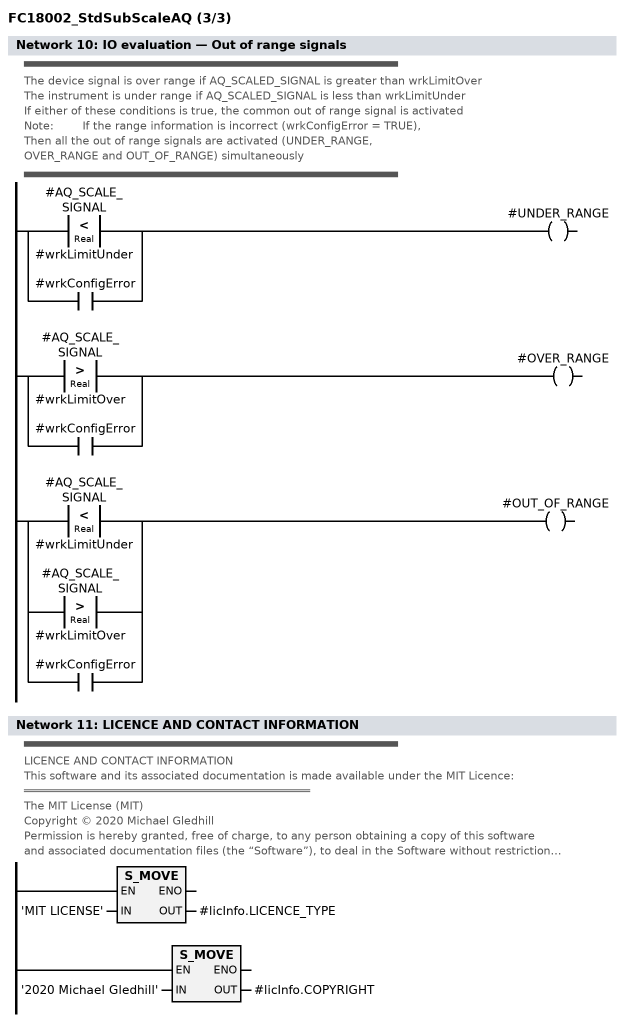
   RUNG wire#powerrail
      { S7_Templates := "SrcType := Real" } LT_Contact(in1 := #AQ_SCALE_SIGNAL, in2 := #wrkLimitUnder)
      wire#w1
      Coil( #UNDER_RANGE )
   END_RUNG
   RUNG wire#powerrail
      Contact( #wrkConfigError )
   END_RUNG wire#w1
   RUNG wire#powerrail
      { S7_Templates := "SrcType := Real" } GT_Contact(in1 := #AQ_SCALE_SIGNAL, in2 := #wrkLimitOver)
      wire#w2
      Coil( #OVER_RANGE )
   END_RUNG
   RUNG wire#powerrail
      Contact( #wrkConfigError )
   END_RUNG wire#w2
   RUNG wire#powerrail
      { S7_Templates := "SrcType := Real" } LT_Contact(in1 := #AQ_SCALE_SIGNAL, in2 := #wrkLimitUnder)
      wire#w3
      Coil( #OUT_OF_RANGE )
   END_RUNG
   RUNG wire#powerrail
      { S7_Templates := "SrcType := Real" } GT_Contact(in1 := #AQ_SCALE_SIGNAL, in2 := #wrkLimitOver)
   END_RUNG wire#w3
   RUNG wire#powerrail
      Contact( #wrkConfigError )
   END_RUNG wire#w3
   // the same network as SCL:
   #UNDER_RANGE := (#AQ_SCALE_SIGNAL < #wrkLimitUnder) OR #wrkConfigError;
   #OVER_RANGE := (#AQ_SCALE_SIGNAL > #wrkLimitOver) OR #wrkConfigError;
   #OUT_OF_RANGE := (#AQ_SCALE_SIGNAL < #wrkLimitUnder) OR (#AQ_SCALE_SIGNAL > #wrkLimitOver) OR #wrkConfigError;
END_REGION

REGION Network 11: LICENCE AND CONTACT INFORMATION
   // ▀▀▀▀▀▀▀▀▀▀▀▀▀▀▀▀▀▀▀▀▀▀▀▀▀▀▀▀▀▀▀▀▀▀▀▀▀▀▀▀▀▀▀▀
   // LICENCE AND CONTACT INFORMATION
   // 
   // This software and its associated documentation is made available under the MIT Licence:
   // 
   // ════════════════════════════════════════════
   // 
   // The MIT License (MIT)
   // 
   // Copyright © 2020 Michael Gledhill
   // 
   // Permission is hereby granted, free of charge, to any person obtaining a copy of this software 
   // and associated documentation files (the “Software”), to deal in the Software without restriction, 
   // including without limitation the rights to use, copy, modify, merge, publish, distribute, 
   // sublicense, and/or sell copies of the Software, and to permit persons to whom the Software is 
   // furnished to do so, subject to the following conditions: 
   // 
   // The above copyright notice and this permission notice shall be included in all copies or 
   // substantial portions of the Software.
   // 
   // THE SOFTWARE IS PROVIDED “AS IS”, WITHOUT WARRANTY OF ANY KIND, EXPRESS OR IMPLIED, 
   // INCLUDING BUT NOT LIMITED TO THE WARRANTIES OF MERCHANTABILITY, FITNESS FOR A 
   // PARTICULAR PURPOSE AND NON-INFRINGEMENT. IN NO EVENT SHALL THE AUTHORS OR COPYRIGHT 
   // HOLDERS BE LIABLE FOR ANY CLAIM, DAMAGES OR OTHER LIABILITY, WHETHER IN AN ACTION OF 
   // CONTRACT, TORT OR OTHERWISE, ARISING FROM, OUT OF OR IN CONNECTION WITH THE SOFTWARE 
   // OR THE USE OR OTHER DEALINGS IN THE SOFTWARE.
   // 
   // ════════════════════════════════════════════
   //                    ┌────────────┐
   // You can reach the author by email here:   │  mg@practicalseries.com  │
   //                    └────────────┘
   // Questions, corrections, constructive criticism and complaints (polite ones) are invited.
   // 
   // ▄▄▄▄▄▄▄▄▄▄▄▄▄▄▄▄▄▄▄▄▄▄▄▄▄▄▄▄▄▄▄▄▄▄▄▄▄▄▄▄▄▄▄▄
   RUNG wire#powerrail
      S_Move(in := 'MIT LICENSE', out => #licInfo.LICENCE_TYPE)
   END_RUNG
   RUNG wire#powerrail
      S_Move(in := '2020 Michael Gledhill', out => #licInfo.COPYRIGHT)
   END_RUNG
   // the same network as SCL:
   #licInfo.LICENCE_TYPE := 'MIT LICENSE';
   #licInfo.COPYRIGHT := '2020 Michael Gledhill';
END_REGION
END_FUNCTION

FUNCTION "FC18151_StdSubTimeEventRTC" : Void   // FC18151, LAD
TITLE = Standard Module [SUBROUTINE] — Event Timer RTC
{ S7_Optimized_Access := 'TRUE' }
AUTHOR : M_Gledhill
FAMILY : Subroutine
NAME : StdSubTimeEventRTC
VERSION : 1.1
// PRACTICAL SERIES AUTOMATION LIBRARY (PAL)   —   COPYRIGHT 2020 – M. GLEDHILL (MIT LICENCE)
//                   ———— ◆ ————
// FULL ONLINE DOCUMENTATION IS AVAILABLE AT: https://practicalseries.com/2001-pal/index.html
// stored: AutoNumber false, IsIECCheckEnabled true, SetENOAutomatically false, UDAEnableTagReadback false
   VAR_INPUT
      TRIGGER : Bool;   // Trigger signal record start time on rising edge, end time on falling edge
   END_VAR
   VAR_IN_OUT
      DYNAMIC_DATA : "UT38151_Dy_SubTimeEventRTC";   // Dynamic data storage (UDT)
   END_VAR
   VAR_TEMP
      revInfo : "UT01000_St_SysRevision";   // Revision information for this block
      licInfo : "UT01001_St_SysLicence";   // Licence information for this block
      wrkInt : Int;   // Working storage area (integer)
      wrkReal : Real;   // Working storage area (real)
      wrkLInt : ULInt;   // Working storage area (long integer, unsigned)
   END_VAR
   VAR_TEMP   // added for the SCL form of the ladder/FBD networks
      _w1 : Bool;
      _w2 : Bool;
   END_VAR
BEGIN

REGION Network 1: Block description — Sections 1 to 3
   // ▄▄▄▄▄▄▄▄▄▄▄▄▄▄▄▄▄▄▄▄▄▄▄▄▄▄▄▄▄▄▄▄▄  ＳＴＡＮＤＡＲＤ  ▄▄ 
   // 
   // 
   // TITLE:    SUBROUTINE — EVENT TIMER RTC
   // 
   // 
   // ▀▀▀▀▀▀▀▀▀▀▀▀▀▀▀▀▀▀▀▀▀▀▀▀▀▀▀▀▀▀▀▀▀▀▀▀▀▀▀▀▀▀▀▀ 
   // 
   // ┌──────────────────────────────────────────┐
   // │                                          │
   // │          FC18151 — SOFTWARE MODULE DESIGN SPECIFICATION (SMDS)            │
   // │                                          │
   // │      The PDF version of the SMDS for this module is available online here:        │
   // │              http://psop.uk/pal-smds-fc18151-p              │
   // │                                          │
   // │      It is also available as part of the Project User Defined Documentation,      │
   // │      it can be accessed by selecting this module in the Project Tree          │
   // │      (on the left) and pressing SHIFT+F1                        │
   // │                                          │
   // └─────────────────────────────────────── ʷᴵᴰ⁻ᵇᵈʰ ┘
   // 
   // FC18151_SubTimeEventRTC is a subroutine block that times the duration of an event 
   // to nanosecond resolution.
   // 
   // The block records the time the event started (rising edge of the TRIGGER signal), the time the 
   // event ended (falling edge of the TRIGGER signal) and calculates the duration of the event (end 
   // time minus the start time).
   // 
   // The start and end times are read from the real time clock of the controller.
   // 
   // This is a subroutine block.
   // 
   // 
   // 
   // ▄▄▄▄▄▄▄▄▄▄▄▄▄▄▄▄▄▄▄▄▄▄▄▄▄▄▄▄▄▄▄▄▄▄▄▄▄▄▄▄▄▄▄▄
   // 1.     BLOCK TECHNICAL SUMMARY
   // 
   // 
   //  ――――――――――――――――――――――――――――――――――――――――――
   //  NOMENCLATURE & ADDRESSING
   //  ――――――――――――――――――――――――――――――――――――――――――
   //  BLOCK TITLE         Subroutine Event Timer using RTC
   //  BLOCK FUNCTION GROUP    Subroutine
   //  BLOCK ADDRESS       FC18151
   //  BLOCK SYMBOL        FC18151_SubTimeEventRTC
   //  BLOCK USER ID         SubTimeEventRTC
   // 
   //  ――――――――――――――――――――――――――――――――――――――――――
   //  BLOCK TYPE & USAGE
   //  ――――――――――――――――――――――――――――――――――――――――――
   //  BLOCK TYPE         Function (FC)
   //  BLOCK NUMBER        18151
   //  LANGUAGE           LAD
   //  OPTIMISED ACCESS     Yes
   //  PAL USAGE TYPE       Standard block
   // 
   //  ――――――――――――――――――――――――――――――――――――――――――
   //  METRICS
   //  ――――――――――――――――――――――――――――――――――――――――――
   //  EXECUTION TIME       18.4 μs¹
   //  LOAD MEMORY       21.4 kB
   //  WORK MEMORY           0.4 kB  
   //  ――――――――――――――――――――――――――――――――――――――――――
   //                ¹ Measured on: CPU-1515-2PN (order no. 6ES7512-2AM02-0AB0) 
   //                             http://psop.uk/pal-ds-cpu1515
   // 
   // 
   // 
   // ▂▂▂▂▂▂▂▂▂▂▂▂▂▂▂▂▂▂▂▂▂▂▂▂▂▂▂▂▂▂▂▂▂▂▂▂▂▂▂▂▂▂▂▂
   // 1.1      Additional document references
   // 
   // 
   // Only those documents specified in OB1 (section DOCUMENT REFERENCES) are listed within this 
   // block. There are no additional document references.
   // 
   //                ━━━   ⬙⬙⬙⬙⬙⬙   ━━━
   // 
   // 
   // 
   // ▄▄▄▄▄▄▄▄▄▄▄▄▄▄▄▄▄▄▄▄▄▄▄▄▄▄▄▄▄▄▄▄▄▄▄▄▄▄▄▄▄▄▄▄
   // 2.     FUNCTIONAL DESCRIPTION
   // 
   // 
   // FC18151 is the Subroutine Event Timer using RTC block, it simply records the duration of an event 
   // with a high degree of accuracy. The event being timed is a Boolean signal passed to the block as 
   // the TRIGGER parameter.
   // 
   // Three times are recorded for the event, the start time (rising edge of the TRIGGER parameter), the 
   // end time (falling edge of the TRIGGER parameter) and the duration of the event (end time minus 
   // the start time). The duration is calculated on the falling edge of the TRIGGER parameter, 
   // immediately after the end time is recorded.
   // 
   // The start and end times are read from the Controller’s internal real time clock (RTC) and are 
   // stored in DTL (date time long) format, this format contains year, month, day, hours, minutes, 
   // seconds, milliseconds, microseconds and nano seconds.
   // 
   // The duration is stored in LTime (long time, 64-bit) format, and is very accurate, it resolves to 
   // days, hours, minutes, seconds milliseconds, microseconds and nanoseconds, it keeps this 
   // resolution irrespective of the duration.
   // 
   // The duration is also calculated as a real number in seconds (or fractions thereof); this is a 
   // more convenient format for holding the duration, but is not as accurate as the LTime format.
   // 
   // 
   // 
   // ▄▄▄▄▄▄▄▄▄▄▄▄▄▄▄▄▄▄▄▄▄▄▄▄▄▄▄▄▄▄▄▄▄▄▄▄▄▄▄▄▄▄▄▄
   // 3.     DETAILED BLOCK DESCRIPTION
   // 
   // The purpose of this block is to determine with a high degree of accuracy the duration of an event, 
   // the event itself must be in the form of a Boolean trigger signal, the rising edge of the signal is 
   // considered to be the start of the event and the falling edge the end of the event.
   // 
   // The event signal is passed to the block as the TRIGGER parameter. 
   // The block returns five values, these are stored in a UDT passed to the block in the 
   // DYNAMIC_DATA parameter: 
   // 
   //  ――――――――――――――――――――――――――――――――――――――――――
   //  PARAM         ASSOCIATED UDT            ASSOCIATED DATA BLOCK
   //  ――――――――――――――――――――――――――――――――――――――――――
   //  DYNAMIC_DATA     UT38151_Dy_SubTimeEventRTC       DB38151_Dy_SubTimeEventRTC
   //  ――――――――――――――――――――――――――――――――――――――――――
   // 
   // 
   // The block returns the following data:
   // 
   //  UT38151_Dy_SubTimeEventRTC
   //  ―――――――――――――――――――――――――――――――――――――――――― 
   //  SIGNAL NAME          FUNCTION                     TYPE
   //  ――――――――――――――――――――――――――――――――――――――――――
   //  status_Running      STATUS — The event timer is running         Bool
   // 
   //  actual_StartTime      ACTUAL — Time at which the TRIGGER signal        DTL
   //                      went high (event start time)
   // 
   //  actual_EndTime        ACTUAL — Time at which the TRIGGER signal     DTL
   //                      went low (event end time)
   // 
   //  actual_Duration        ACTUAL — Event duration              LTime
   // 
   //  actual_DurationSec       ACTUAL — Event duration in seconds           REAL
   //  ――――――――――――――――――――――――――――――――――――――――――
   // 
   // 
   // 
   // ▂▂▂▂▂▂▂▂▂▂▂▂▂▂▂▂▂▂▂▂▂▂▂▂▂▂▂▂▂▂▂▂▂▂▂▂▂▂▂▂▂▂▂▂
   // 3.1     Timing an event
   // 
   // The block constantly monitors the TRIGGER parameter; if a rising edge is seen on the TRIGGER 
   // parameter (point ① in the figure below), the Controller RTC is read and its value is stored in 
   // actual_StartTime, at the same time the running signal (status_Running) is activated.
   // 
   // The block continues to monitor the TRIGGER parameter, when a falling edge is detected 
   // (point ②), the RTC is read once more and its value is stored in actual_EndTime, and the running 
   // signal (status_Running) is deactivated.
   // 
   // Once the end time is stored, the following calculation is carried out:
   // 
   // 
   // ┌───────────────────────────┐
   // │ actual_Duration =  actual_EndTime ─ actual_StartTime    │
   // └───────────────────────────┘
   // 
   // 
   //                     ①            ②
   //   TRIGGER │             ┏━━━━━━━━━━━━┓
   //         │             ┃               ┃
   //         │             ┃               ┃
   //         │             ┃               ┃
   //         │             ┃               ┃                              
   //         ┼━━━━━━━━━━━━╶╶╶╶╶╶╶╶╶╶╶╶╶━━━━━━━━━━ time
   //                  ↗             ↖
   //          actual_Start_Time ╎            ╎ actual_End_Time
   //    DTL#2020-04-18-09:34:25.899548353        DTL#2020-04-18-09:34:36.004744916
   // 
   //                    ╎               ╎                      actual_Duration
   //                                      LT#10S_105MS_196US_563NS
   //                    ╎               ╎  
   //                                                     actual_DurationSec
   //                    ╎               ╎                              10.10519
   // 
   //         │status_Running      ┏━━━━━━━━━━━━┓
   //         │             ┃               ┃
   //         │             ┃               ┃
   //         │             ┃               ┃
   //         │             ┃               ┃
   //         ┼━━━━━━━━━━━━╶╶╶╶╶╶╶╶╶╶╶╶╶━━━━━━━━━━
   // 
   // 
   // 
   // ▂▂▂▂▂▂▂▂▂▂▂▂▂▂▂▂▂▂▂▂▂▂▂▂▂▂▂▂▂▂▂▂▂▂▂▂▂▂▂▂▂▂▂▂
   // 3.1     Date and time data types
   // 
   // Both the start and end times (actual_StartTime and actual_EndTime) are of the type DTL 
   // (date time long), this itself is a data structure in the form:
   // 
   //  DTL Data Structure
   //  ――――――――――――――――――――――――――――――――――――――――――
   //  SIGNAL NAME          FUNCTION                     TYPE
   //  ――――――――――――――――――――――――――――――――――――――――――
   //  YEAR             Year (returns a value in the range 1970 to 2262)     UInt
   //  MONTH            Month (1-12 representing Jan to Dec)        USInt
   //  DAY              Day of month (1-31)                USInt
   //  WEEKDAY          Day of week (1-7, where 1=Sunday, 7=Saturday)    USInt
   //  HOUR           Hour of day (0-23)                   USInt
   //  MINUTE           Minutes (0-59)                   USInt
   //  SECOND            Seconds (0-59)                  USInt
   //  NANOSECOND        Nanoseconds (0-999,999,999)           UDint
   //  ――――――――――――――――――――――――――――――――――――――――――
   // 
   // When displayed, it has the format:
   // 
   //       DTL#2020-04-18-09:34:25.899548353
   // 
   //  I.e.      18th April 2020 at 09:43:25 AM and 899,548,353 ns.
   // 
   // The calculated duration (actual_Duration) is of data type LTime (long time).
   // 
   // The LTime data type is essentially an 8-byte number (64-bit number) that stores a time value in 
   // nanoseconds. In the above example, the actual_Duration has the formatted value of:
   // 
   //       LT#10S_105MS_196US_563NS
   // 
   //  I.e.      10 seconds, 105 milliseconds, 196 microseconds and 563 nanoseconds.
   // 
   // It is shown in this format, because TIA portal understands the LTime data type and is able to 
   // interpret the value as days, hours, minute, seconds, milliseconds, microseconds and 
   // nanoseconds. 
   // 
   // In practice, the actual_Duration simply (in this example) holds a very large number:
   // 
   //       10,105,196,563
   // 
   // This is the duration of the event in nanoseconds (i.e. 10,105,196,563 nanoseconds). To convert 
   // the number to seconds, simply divide by 1,000,000,000 (or 1 × 10^9); this would give:
   // 
   //       10.105196563 seconds
   // 
   // The reason the duration is specified as an LTime rather that DTL is that, somewhat confusingly, 
   // DTL is a relative measure of time (relative to 1st January, 1970), if the above duration were 
   // represented as a DTL value it would read:
   // 
   //       DTL#1970-01-01-00:00:10.105196563
   // 
   // Hours, minutes and seconds are OK, but the date part doesn’t make sense (to make it 
   // meaningful, 1970 must be subtracted from the YEAR value and 1 from both the MONTH and 
   // DAY values).
   // 
   // The LTime data type can store a duration of up to 106,751 days (about 300 years) and while not 
   // perfect, it seems long enough for most practical situations (possibly not for geological 
   // applications).
   // 
   // The actual_Duration in LTime format is very accurate, but it is an unwieldly data type, to provide a 
   // more user friendly (although less accurate) format, the actual_Duration signal is converted to a 
   // real number giving the duration in seconds, this is stored in the actual_DurationSec signal. In the 
   // above example: 
   // 
   //       actual_DurationSec has the value 10.10519 seconds
   // 
   // It is less accurate, it does not resolve to nanoseconds; however, it is easier to use and display 
   // and is accurate enough for most applications.
   // 
   // 
   // 
   // ▁▁▁▁▁▁▁▁▁▁▁▁▁▁▁▁▁▁▁▁▁▁▁▁▁▁▁▁▁▁▁▁▁▁▁▁▁▁▁▁▁▁▁▁
   // A note on real numbers (and accuracy)
   // 
   // The LTime format is very accurate, it is basically counting nanoseconds, and because it is 64-bits 
   // long it can count up to very high values (about 292 years at nanosecond resolution).
   // 
   // Real numbers however, are limited to 32-bits and suffer from precision loss, this results from the 
   // fact that the real number has an accuracy of “about” 7 decimal digits, for example 20365.45, 
   // 20.43728, 1.482967, 0.3356428, &c. Essentially, the bigger the number, the fewer the decimal 
   // places — a total of 7 decimal digits.
   // 
   // Very big and very small numbers can be represented by adding trailing zeros for big numbers 
   // (e.g. 3275625000) and leading zeros for small numbers (0.000003275625) in both these 
   // examples, there are only 7 decimal digits, just shifted effectively left or right.
   // 
   // This type of representation is usually handled by applying scientific notation, the number 
   // 1,568,497,000,000 would be represented as 1.568497 × 10^12, it only has 7 decimal digits, 
   // the number 1,568,497,132,792, would be represented as exactly the same value, the 132,792 
   // part of the number can not be resolved and are lost.
   // 
   //                ━━━   ⬙⬙⬙⬙⬙⬙   ━━━
   // 
   // 
   // 
   // ▄▄▄▄▄▄▄▄▄▄▄▄▄▄▄▄▄▄▄▄▄▄▄▄▄▄▄▄▄▄▄▄▄▄▄▄▄▄▄▄▄▄▄▄
   // 4.     Supervisory system interface
   // 
   // 
   // FC18151 is a Subroutine block. It does not have a supervisory system interface.
   // 
   // 
   //                ━━━   ⬙⬙⬙⬙⬙⬙   ━━━
   // 
   // 
   // 
   // ▄▄▄▄▄▄▄▄▄▄▄▄▄▄▄▄▄▄▄▄▄▄▄▄▄▄▄▄▄▄▄▄▄▄▄▄▄▄▄▄▄▄▄▄
   // 5.     PARAMETERS
   // 
   // 
   // The following parameters are associated with the block:
   // 
   //  
   //  ――――――――――――――――――――――――――――――――――――――――――
   //  PARAM         FUNCTION                    TYPE      IN-OUT 
   //  ――――――――――――――――――――――――――――――――――――――――――
   //  TRIGGER       Event trigger signal (a rising edge marks the     Bool   In
   //           start of the event, the falling edge the end)
   // 
   // 
   //  DYNAMIC_DATA      Stores the results of the event timing       UT38151    InOut
   //  ――――――――――――――――――――――――――――――――――――――――――
   // 
   // Note:    FC18151 is one of the few blocks that does not require the SYS_SIGNALS parameter 
   //      (this has been done to make minimise the block interface)
   // 
   //                ━━━   ⬙⬙⬙⬙⬙⬙   ━━━
   // 
   // 
   // 
   // ▄▄▄▄▄▄▄▄▄▄▄▄▄▄▄▄▄▄▄▄▄▄▄▄▄▄▄▄▄▄▄▄▄▄▄▄▄▄▄▄▄▄▄▄
   // 6.     DATA STRUCTURES AND USAGE
   // 
   // 
   // The block has the following associated data structure:
   // 
   // 
   //  ――――――――――――――――――――――――――――――――――――――――――
   //  DATA STRUCTURE             DESCRIPTION
   //  ――――――――――――――――――――――――――――――――――――――――――
   //  UT01000_St_SysRevision          Revision information for this block    See FC01001
   //  UT01001_St_SysLicence           Licence information for this block  See FC01001
   //  UT38151_Dy_SubTimeEventRTC        Dynamic data structure for the event timing block
   //  ――――――――――――――――――――――――――――――――――――――――――
   // 
   // 
   // 
   // ▂▂▂▂▂▂▂▂▂▂▂▂▂▂▂▂▂▂▂▂▂▂▂▂▂▂▂▂▂▂▂▂▂▂▂▂▂▂▂▂▂▂▂▂
   // 6.1     UT38151_Dy_TimeEventRTC
   // 
   // Stores the timing values for the event:
   // 
   //  UT38151_Dy_TimeEventRTC
   //  ――――――――――――――――――――――――――――――――――――――――――
   //  SIGNAL NAME          FUNCTION                     TYPE
   //  ――――――――――――――――――――――――――――――――――――――――――
   //  status_Running      STATUS — The event timer is running         Bool
   // 
   //  actual_StartTime      ACTUAL — Time at which the TRIGGER signal        DTL
   //                      went high (event start time)
   // 
   //  actual_EndTime        ACTUAL — Time at which the TRIGGER signal     DTL
   //                      went low (event end time)
   // 
   //  actual_Duration        ACTUAL — Event duration              LTime
   // 
   //  actual_DurationSec       ACTUAL — Event duration in seconds           REAL
   //  ――――――――――――――――――――――――――――――――――――――――――
   // 
   //                ━━━   ⬙⬙⬙⬙⬙⬙   ━━━
   // 
   // 
   // 
   // ▄▄▄▄▄▄▄▄▄▄▄▄▄▄▄▄▄▄▄▄▄▄▄▄▄▄▄▄▄▄▄▄▄▄▄▄▄▄▄▄▄▄▄▄
   // 7.     CONSTANTS AND TEMPORARY (LOCAL) DATA
   // 
   // 
   // 
   // ▂▂▂▂▂▂▂▂▂▂▂▂▂▂▂▂▂▂▂▂▂▂▂▂▂▂▂▂▂▂▂▂▂▂▂▂▂▂▂▂▂▂▂▂
   // 7.1     Constants
   // 
   // 
   // No constants are used in this block.
   // 
   // 
   // 
   // ▂▂▂▂▂▂▂▂▂▂▂▂▂▂▂▂▂▂▂▂▂▂▂▂▂▂▂▂▂▂▂▂▂▂▂▂▂▂▂▂▂▂▂▂
   // 7.2     Temporary (local) data
   // 
   // 
   // The following temporary data is used:
   // 
   //  ――――――――――――――――――――――――――――――――――――――――――
   //  SIGNAL NAME          FUNCTION                  TYPE
   //  ――――――――――――――――――――――――――――――――――――――――――
   //  revInfo             Revision information for the block         UT01000
   //  licInfo           Licensing information for the block      UT01001
   //  wrkInt           Working storage area (integer)          Int
   //  wrkReal           Working storage (Real)             Real
   //  wrkLInt            Working storage area (longinteger)      LInt
   //  ――――――――――――――――――――――――――――――――――――――――――
   // 
   //                ━━━   ⬙⬙⬙⬙⬙⬙   ━━━
   // 
   // 
   // 
   // ▄▄▄▄▄▄▄▄▄▄▄▄▄▄▄▄▄▄▄▄▄▄▄▄▄▄▄▄▄▄▄▄▄▄▄▄▄▄▄▄▄▄▄▄
   // 8.     BLOCK CALLS AND ASSOCIATIONS
   // 
   // 
   // This section details any blocks which may be called from within this software module (subroutine 
   // functions for example), any partner blocks with which it may be associated (for example a 
   // receive module that is partner with a transmit module &c.). It lists any system functions which 
   // may be called (e.g. reading the real time clock) and any system data types that may be used.
   // 
   // Finally, it lists any special calling requirements for the block (for example, must be called from 
   // within a cyclic interrupt organisation block) and if the block is using “optimised access” (this is 
   // the default arrangement).
   // 
   // 
   // 
   // ▂▂▂▂▂▂▂▂▂▂▂▂▂▂▂▂▂▂▂▂▂▂▂▂▂▂▂▂▂▂▂▂▂▂▂▂▂▂▂▂▂▂▂▂
   // 8.1     Block calls from within this module
   // 
   // 
   // There are no PAL block calls from within this block.
   // 
   // 
   // 
   // ▂▂▂▂▂▂▂▂▂▂▂▂▂▂▂▂▂▂▂▂▂▂▂▂▂▂▂▂▂▂▂▂▂▂▂▂▂▂▂▂▂▂▂▂
   // 8.2     Blocks associated with this module
   // 
   // 
   // This is a stand-alone block and is not associated with any other blocks.
   // 
   // 
   // 
   // ▂▂▂▂▂▂▂▂▂▂▂▂▂▂▂▂▂▂▂▂▂▂▂▂▂▂▂▂▂▂▂▂▂▂▂▂▂▂▂▂▂▂▂▂
   // 8.3     System block calls and system data typesThe following calls are made to system blocks:
   // 
   // 
   //  System block calls
   //  ――――――――――――――――――――――――――――――――――――――――――
   //  BLOCK          TITLE             DESCRIPTION  
   //  ――――――――――――――――――――――――――――――――――――――――――
   //  RD_LOC_T             Read the local RTC time    Reads the CPU real time clock 
   //  ――――――――――――――――――――――――――――――――――――――――――
   // 
   // There are no special system data types used.
   // 
   // 
   // 
   // ▂▂▂▂▂▂▂▂▂▂▂▂▂▂▂▂▂▂▂▂▂▂▂▂▂▂▂▂▂▂▂▂▂▂▂▂▂▂▂▂▂▂▂▂
   // 8.4     Special properties and requirements
   // 
   // 
   // 
   // ▁▁▁▁▁▁▁▁▁▁▁▁▁▁▁▁▁▁▁▁▁▁▁▁▁▁▁▁▁▁▁▁▁▁▁▁▁▁▁▁▁▁▁▁
   // 8.4.1     Block optimisation, IEC compatibility and library conformance
   // 
   // 
   //    •   Block optimisation is ACTIVE for this block.
   // 
   //    •   The block has been checked for IEC compatibility and is compliant.
   // 
   //    •   The block is compatible with all IEC library-conformance module constraints
   // 
   // 
   // 
   // ▁▁▁▁▁▁▁▁▁▁▁▁▁▁▁▁▁▁▁▁▁▁▁▁▁▁▁▁▁▁▁▁▁▁▁▁▁▁▁▁▁▁▁▁
   // 8.4.2     Calling requirements
   // 
   // 
   // There are no special calling requirements for this block.
   // 
   //                ━━━   ⬙⬙⬙⬙⬙⬙   ━━━
   // 
   // 
   // 
   // ▄▄▄▄▄▄▄▄▄▄▄▄▄▄▄▄▄▄▄▄▄▄▄▄▄▄▄▄▄▄▄▄▄▄▄▄▄▄▄▄▄▄▄▄
   // 9.     EXAMPLE USAGE
   // 
   // 
   // The following shows a typical deployment of FC18151:
   // 
   //                      ┌─────────────
   //        ──────────────┤ FC18151
   //                      ├───────────
   //                 %M100.0    │
   //               "Event001"   ─┤ TRIGGER
   //                      │
   //     "DB38151_Dy_TimeEventRTC".Event001 ─┤ DYNAMIC_DATA
   //                      │
   //                      │             │
   //                                    │
   //                           ─────────┘
   // 
   //               ━━━   ⬙⬙⬙⬙⬙⬙   ━━━
   // 
   // 
   // 
   // ▄▄▄▄▄▄▄▄▄▄▄▄▄▄▄▄▄▄▄▄▄▄▄▄▄▄▄▄▄▄▄▄▄▄▄▄▄▄▄▄▄▄▄▄
   // 10.     TEST AND VERIFICATION PATH
   // 
   // 
   // The following diagram shows the full test and verification path for the formal release of each 
   // version of the software module. See the Test Plan [Ref. 003] for full details, available here:
   //         http://psop.uk/pal-tp-p
   // 
   // 
   //         FC18151-T001         FC18151-T002
   // 
   //     Test version: 000.801     Test version: 001.801
   //  Released version: 001.000     Released version: 002.000
   // Released commit: D0003    Released commit: D0011
   // 
   //        SCR      SMT              SCV     
   // ＿＿＿＿＿＿┌┐＿＿ ▛▜ ＿＿＿＿＿＿＿＿＿＿＿＿╓╖＿＿
   //       └┘   ▙▟             ╙╜  
   // Initial test           Comments standardised
   // 
   // Initial test to release the      Comments updated & 
   // module following the      minor typographical 
   // development stage.       corrections
   // Full SMT              SCV only
   // 
   // 
   // Where:
   // ――――――――――――――――――――――――――――――――――――――――――――
   //  SCR    Source Code Review      A visual inspection of the software to ensure it has been written  
   // ┌┐             to the correct standards, uses the correct structures within the
   // └┘             software and is generally suitable for deployment.               
   // 
   //  SMT Software Module Test    A full and detailed test of an individual software module in
   //   ▛▜              isolation; such testing requires that all branches of the 
   //   ▙▟              software are tested. 
   // 
   //                It tests all the interfaces to the module, any data recorded or 
   //                stored by the module, all error and exception handling functions 
   //                and tests all timed and interrupt driven operations.
   // 
   //  SCV Software Compatibility     A mechanism for verifying that no executable code software 
   // ╓╖    Verification          changes have been made to a module following changes to
   // ╙╜             comment fields.
   // 
   //                Allows typographical errors &c. to be corrected without forcing 
   //                a full SMT on a module that has not functionally changed.
   // ――――――――――――――――――――――――――――――――――――――――――――
   // 
   // An SCV can only be performed on a module that has at some point previously, successfully 
   // completed both an SCR and SMT. Where an SCV is implemented, it replaces the requirement for 
   // both the SCR and the SMT for the test iteration in question.
   // 
   //                ━━━   ⬙⬙⬙⬙⬙⬙   ━━━
   // 
   // 
   // 
   // ██████████████ █ █ █ █  END   █ █ █ █ ██████████████
END_REGION

REGION Network 2: Current revision and modification history
   // ▄▄▄▄▄▄▄▄▄▄▄▄▄▄▄▄▄▄▄▄▄▄▄▄▄▄▄▄▄▄▄▄▄▄▄▄▄▄▄▄▄▄▄▄
   // MODIFICATION HISTORY
   // 
   // 
   // The revision data shown here, in the network comments, contains additional information 
   // reflecting the software development workflow under the version control system (VCS) employed 
   // to track all software changes.
   // 
   // The VCS in use is the Git Source Code Management system in conjunction with the GitHub online 
   // hosting system. The software in its entirety is available in the GitHub remote repository:
   // 
   //      https://github.com/practicalseries/PS2001-pal-software
   // 
   // The repository is public and can be freely copied (forked in GitHub terminology) and used 
   // under the MIT licence. 
   // 
   // The MIT licence is reproduced in full in the last network of this software module
   // 
   // 
   //  ―――――――――――――――――――――――――――――――――――――――――――
   //  DATE       REVISION             MASTER BRANCH     DEV
   //          (nnn.amm)   COMMIT TAG    (Base ---> Merge)    BRANCH   Author
   //  ———————————————————————————————————————————
   //  2022.04.08    001.101   D0010A-000.104   D0010 N/A     D010A   M. Gledhill
   //                        Comments updated and standardised
   //                        NW 2 comments combined with NW 1
   // 
   //  2021.02.19    001.000   D0003      D0002 D0003  None    M. Gledhill
   //                        FC18151 — RELEASED FOR USE
   //                          Merge back to master branch
   // 
   //  2021.02.19    001.000   D0002A-001.000   D0002 N/A     D0002A   M. Gledhill
   //                        FC18151 — Post test RELEASED FOR USE
   //  
   //  2021.02.18    000.801   D0002A-000.801   D0002 N/A     D0002A   M. Gledhill
   //                        FC18151 Migration to VCS — Released for test
   //  ———————————————————————————————————————————
   //   Where: nnn  =  Major revision
   //         a  =  Type (1-7 Development, 8 Proving, 9 Qualification, 0 Release)
   //       mm  =  Minor revision (must be 00 if a = 0)
   //         Block properties version number should be set to nn.a (only one decimal place)
   // 
   // ▄▄▄▄▄▄▄▄▄▄▄▄▄▄▄▄▄▄▄▄▄▄▄▄▄▄▄▄▄▄▄▄▄▄▄▄▄▄▄▄▄▄▄▄
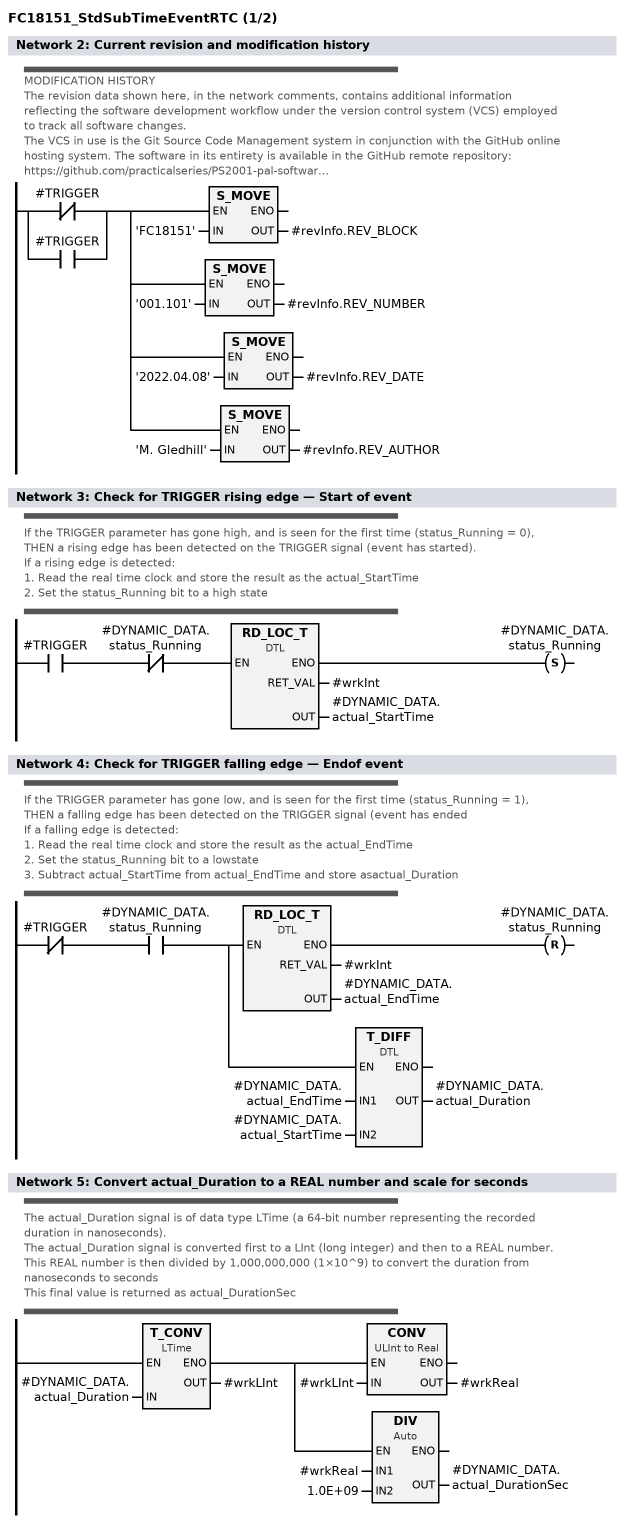
   RUNG wire#powerrail
      I_Contact( #TRIGGER )
      wire#w1
      S_Move(in := 'FC18151', out => #revInfo.REV_BLOCK)
   END_RUNG
   RUNG wire#powerrail
      Contact( #TRIGGER )
   END_RUNG wire#w1
   RUNG wire#w1
      S_Move(in := '001.101', out => #revInfo.REV_NUMBER)
   END_RUNG
   RUNG wire#w1
      S_Move(in := '2022.04.08', out => #revInfo.REV_DATE)
   END_RUNG
   RUNG wire#w1
      S_Move(in := 'M. Gledhill', out => #revInfo.REV_AUTHOR)
   END_RUNG
   // the same network as SCL:
   IF NOT #TRIGGER OR #TRIGGER THEN
       #revInfo.REV_BLOCK := 'FC18151';
       #revInfo.REV_NUMBER := '001.101';
       #revInfo.REV_DATE := '2022.04.08';
       #revInfo.REV_AUTHOR := 'M. Gledhill';
   END_IF;
END_REGION

REGION Network 3: Check for TRIGGER rising edge — Start of event
   // ▀▀▀▀▀▀▀▀▀▀▀▀▀▀▀▀▀▀▀▀▀▀▀▀▀▀▀▀▀▀▀▀▀▀▀▀▀▀▀▀▀▀▀▀
   // If the TRIGGER parameter has gone high, and is seen for the first time (status_Running = 0),
   // THEN a rising edge has been detected on the TRIGGER signal (event has started).
   // 
   // If a rising edge is detected:
   //   1. Read the real time clock and store the result as the actual_StartTime
   //   2. Set the status_Running bit to a high state
   // ▄▄▄▄▄▄▄▄▄▄▄▄▄▄▄▄▄▄▄▄▄▄▄▄▄▄▄▄▄▄▄▄▄▄▄▄▄▄▄▄▄▄▄▄
   RUNG wire#powerrail
      Contact( #TRIGGER )
      I_Contact( #DYNAMIC_DATA.status_Running )
      { S7_Templates := "date_type := DTL" } RD_LOC_T(RET_VAL => #wrkInt, OUT => #DYNAMIC_DATA.actual_StartTime)
      S_Coil( #DYNAMIC_DATA.status_Running )
   END_RUNG
   // the same network as SCL:
   #wrkInt := RD_LOC_T(EN := #TRIGGER AND NOT #DYNAMIC_DATA.status_Running,
                       OUT => #DYNAMIC_DATA.actual_StartTime,
                       ENO => #_w1);
   IF #_w1 THEN #DYNAMIC_DATA.status_Running := TRUE; END_IF;
END_REGION

REGION Network 4: Check for TRIGGER falling edge — Endof event
   // ▀▀▀▀▀▀▀▀▀▀▀▀▀▀▀▀▀▀▀▀▀▀▀▀▀▀▀▀▀▀▀▀▀▀▀▀▀▀▀▀▀▀▀▀
   // If the TRIGGER parameter has gone low, and is seen for the first time (status_Running = 1),
   // THEN a falling edge has been detected on the TRIGGER signal (event has ended
   // 
   // If a falling edge is detected:
   //   1. Read the real time clock and store the result as the actual_EndTime
   //   2. Set the status_Running bit to a lowstate
   //   3. Subtract actual_StartTime from actual_EndTime and store asactual_Duration
   // ▄▄▄▄▄▄▄▄▄▄▄▄▄▄▄▄▄▄▄▄▄▄▄▄▄▄▄▄▄▄▄▄▄▄▄▄▄▄▄▄▄▄▄▄
   RUNG wire#powerrail
      I_Contact( #TRIGGER )
      Contact( #DYNAMIC_DATA.status_Running )
      wire#w1
      { S7_Templates := "date_type := DTL" } RD_LOC_T(RET_VAL => #wrkInt, OUT => #DYNAMIC_DATA.actual_EndTime)
      R_Coil( #DYNAMIC_DATA.status_Running )
   END_RUNG
   RUNG wire#w1
      { S7_Templates := "[date_type := DTL, time_type := LTime]" } T_DIFF(IN1 := #DYNAMIC_DATA.actual_EndTime, IN2 := #DYNAMIC_DATA.actual_StartTime, OUT => #DYNAMIC_DATA.actual_Duration)
   END_RUNG
   // the same network as SCL:
   #wrkInt := RD_LOC_T(EN := NOT #TRIGGER AND #DYNAMIC_DATA.status_Running,
                       OUT => #DYNAMIC_DATA.actual_EndTime,
                       ENO => #_w1);
   #_w2 := NOT #TRIGGER AND #DYNAMIC_DATA.status_Running;
   IF #_w1 THEN #DYNAMIC_DATA.status_Running := FALSE; END_IF;
   IF #_w2 THEN
       T_DIFF(IN1 := #DYNAMIC_DATA.actual_EndTime,
              IN2 := #DYNAMIC_DATA.actual_StartTime,
              OUT => #DYNAMIC_DATA.actual_Duration);
   END_IF;
END_REGION

REGION Network 5: Convert actual_Duration to a REAL number and scale for seconds
   // ▀▀▀▀▀▀▀▀▀▀▀▀▀▀▀▀▀▀▀▀▀▀▀▀▀▀▀▀▀▀▀▀▀▀▀▀▀▀▀▀▀▀▀▀
   // The actual_Duration signal is of data type LTime (a 64-bit number representing the recorded
   // duration in nanoseconds).
   // 
   // The actual_Duration signal is converted first to a LInt (long integer) and then to a REAL number.
   // 
   // This REAL number is then divided by 1,000,000,000 (1×10^9) to convert the duration from 
   // nanoseconds to seconds
   // 
   // This final value is returned as actual_DurationSec
   // ▄▄▄▄▄▄▄▄▄▄▄▄▄▄▄▄▄▄▄▄▄▄▄▄▄▄▄▄▄▄▄▄▄▄▄▄▄▄▄▄▄▄▄▄
   RUNG wire#powerrail
      { S7_Templates := "[src_type := LTime, dest_type := ULInt]" } T_CONV(IN := #DYNAMIC_DATA.actual_Duration, OUT => #wrkLInt)
      wire#w1
      { S7_Templates := "[SrcType := ULInt, DestType := Real]" } Convert(in := #wrkLInt, out => #wrkReal)
   END_RUNG
   RUNG wire#w1
      Div(in1 := #wrkReal, in2 := 1.0E+09, out => #DYNAMIC_DATA.actual_DurationSec)
   END_RUNG
   // the same network as SCL:
   T_CONV(IN := #DYNAMIC_DATA.actual_Duration, OUT => #wrkLInt, ENO => #_w1);
   IF #_w1 THEN
       #wrkReal := ULINT_TO_REAL(#wrkLInt);
       #DYNAMIC_DATA.actual_DurationSec := #wrkReal / 1.0E+09;
   END_IF;
END_REGION

REGION Network 6: LICENCE AND CONTACT INFORMATION
   // ▀▀▀▀▀▀▀▀▀▀▀▀▀▀▀▀▀▀▀▀▀▀▀▀▀▀▀▀▀▀▀▀▀▀▀▀▀▀▀▀▀▀▀▀
   // LICENCE AND CONTACT INFORMATION
   // 
   // This software and its associated documentation is made available under the MIT Licence:
   // 
   // ════════════════════════════════════════════
   // 
   // The MIT License (MIT)
   // 
   // Copyright © 2020 Michael Gledhill
   // 
   // Permission is hereby granted, free of charge, to any person obtaining a copy of this software 
   // and associated documentation files (the “Software”), to deal in the Software without restriction, 
   // including without limitation the rights to use, copy, modify, merge, publish, distribute, 
   // sublicense, and/or sell copies of the Software, and to permit persons to whom the Software is 
   // furnished to do so, subject to the following conditions: 
   // 
   // The above copyright notice and this permission notice shall be included in all copies or 
   // substantial portions of the Software.
   // 
   // THE SOFTWARE IS PROVIDED “AS IS”, WITHOUT WARRANTY OF ANY KIND, EXPRESS OR IMPLIED, 
   // INCLUDING BUT NOT LIMITED TO THE WARRANTIES OF MERCHANTABILITY, FITNESS FOR A 
   // PARTICULAR PURPOSE AND NON-INFRINGEMENT. IN NO EVENT SHALL THE AUTHORS OR COPYRIGHT 
   // HOLDERS BE LIABLE FOR ANY CLAIM, DAMAGES OR OTHER LIABILITY, WHETHER IN AN ACTION OF 
   // CONTRACT, TORT OR OTHERWISE, ARISING FROM, OUT OF OR IN CONNECTION WITH THE SOFTWARE 
   // OR THE USE OR OTHER DEALINGS IN THE SOFTWARE.
   // 
   // ════════════════════════════════════════════
   //                    ┌────────────┐
   // You can reach the author by email here:   │  mg@practicalseries.com  │
   //                    └────────────┘
   // Questions, corrections, constructive criticism and complaints (polite ones) are invited.
   // 
   // ▄▄▄▄▄▄▄▄▄▄▄▄▄▄▄▄▄▄▄▄▄▄▄▄▄▄▄▄▄▄▄▄▄▄▄▄▄▄▄▄▄▄▄▄
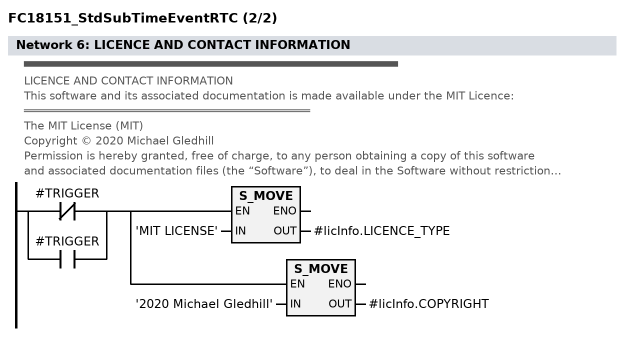
   RUNG wire#powerrail
      I_Contact( #TRIGGER )
      wire#w1
      S_Move(in := 'MIT LICENSE', out => #licInfo.LICENCE_TYPE)
   END_RUNG
   RUNG wire#powerrail
      Contact( #TRIGGER )
   END_RUNG wire#w1
   RUNG wire#w1
      S_Move(in := '2020 Michael Gledhill', out => #licInfo.COPYRIGHT)
   END_RUNG
   // the same network as SCL:
   IF NOT #TRIGGER OR #TRIGGER THEN
       #licInfo.LICENCE_TYPE := 'MIT LICENSE';
       #licInfo.COPYRIGHT := '2020 Michael Gledhill';
   END_IF;
END_REGION
END_FUNCTION

DATA_BLOCK "Timer_day"   // DB5
{ S7_Optimized_Access := 'TRUE' }
// stored: AutoNumber false, DBAccessibleFromOPCUA true, InstanceOfName IEC_TIMER, OfSystemLibElement IEC_TIMER, OfSystemLibVersion 1.0
"IEC_TIMER"
   // VAR
   //    PT : Time;
   //    ET { ExternalWritable := 'False'} : Time;
   //    IN : Bool;
   //    Q { ExternalWritable := 'False'} : Bool;
   // END_VAR
BEGIN
END_DATA_BLOCK

DATA_BLOCK "Timer_hour"   // DB4
{ S7_Optimized_Access := 'TRUE' }
// stored: AutoNumber false, DBAccessibleFromOPCUA true, InstanceOfName IEC_TIMER, OfSystemLibElement IEC_TIMER, OfSystemLibVersion 1.0
"IEC_TIMER"
   // VAR
   //    PT : Time;
   //    ET { ExternalWritable := 'False'} : Time;
   //    IN : Bool;
   //    Q { ExternalWritable := 'False'} : Bool;
   // END_VAR
BEGIN
END_DATA_BLOCK

DATA_BLOCK "Timer_min"   // DB3
{ S7_Optimized_Access := 'TRUE' }
// stored: AutoNumber false, DBAccessibleFromOPCUA true, InstanceOfName IEC_TIMER, OfSystemLibElement IEC_TIMER, OfSystemLibVersion 1.0
"IEC_TIMER"
   // VAR
   //    PT : Time;
   //    ET { ExternalWritable := 'False'} : Time;
   //    IN : Bool;
   //    Q { ExternalWritable := 'False'} : Bool;
   // END_VAR
BEGIN
END_DATA_BLOCK

DATA_BLOCK "Timer_ms"   // DB1
{ S7_Optimized_Access := 'TRUE' }
// stored: AutoNumber true, DBAccessibleFromOPCUA true, InstanceOfName IEC_TIMER, OfSystemLibElement IEC_TIMER, OfSystemLibVersion 1.0
"IEC_TIMER"
   // VAR
   //    PT : Time;
   //    ET { ExternalWritable := 'False'} : Time;
   //    IN : Bool;
   //    Q { ExternalWritable := 'False'} : Bool;
   // END_VAR
BEGIN
END_DATA_BLOCK

DATA_BLOCK "Timer_sec"   // DB2
{ S7_Optimized_Access := 'TRUE' }
// stored: AutoNumber false, DBAccessibleFromOPCUA true, InstanceOfName IEC_TIMER, OfSystemLibElement IEC_TIMER, OfSystemLibVersion 1.0
"IEC_TIMER"
   // VAR
   //    PT : Time;
   //    ET { ExternalWritable := 'False'} : Time;
   //    IN : Bool;
   //    Q { ExternalWritable := 'False'} : Bool;
   // END_VAR
BEGIN
END_DATA_BLOCK
